C01810=1171.717,232.946,-63.644,-177.541,7.223,148.639
C01811=1171.722,232.698,-63.619,-177.544,7.221,148.640
C01812=1171.727,232.450,-63.593,-177.547,7.218,148.640
C01813=1171.731,232.200,-63.567,-177.549,7.216,148.640
C01814=1171.736,231.952,-63.541,-177.552,7.214,148.640
C01815=1171.740,231.703,-63.515,-177.555,7.211,148.640
C01816=1171.744,231.455,-63.489,-177.557,7.209,148.640
C01817=1171.749,231.207,-63.464,-177.560,7.206,148.640
C01818=1171.754,230.957,-63.437,-177.563,7.204,148.641
C01819=1171.758,230.709,-63.411,-177.566,7.201,148.641
C01820=1171.762,230.460,-63.386,-177.568,7.199,148.641
C01821=1171.767,230.212,-63.360,-177.571,7.196,148.641
C01822=1171.771,229.963,-63.335,-177.573,7.194,148.641
C01823=1171.775,229.714,-63.309,-177.576,7.192,148.642
C01824=1171.780,229.465,-63.282,-177.579,7.190,148.642
C01825=1171.785,229.217,-63.257,-177.581,7.187,148.642
C01826=1171.789,228.968,-63.231,-177.584,7.185,148.642
C01827=1171.794,228.719,-63.206,-177.587,7.182,148.642
C01828=1171.798,228.471,-63.180,-177.590,7.179,148.643
C01829=1171.803,228.222,-63.154,-177.592,7.177,148.643
C01830=1171.807,227.974,-63.129,-177.595,7.175,148.643
C01831=1171.812,227.725,-63.103,-177.598,7.172,148.643
C01832=1171.816,227.477,-63.078,-177.601,7.170,148.643
C01833=1171.820,227.228,-63.052,-177.603,7.168,148.644
C01834=1171.825,226.980,-63.026,-177.606,7.165,148.644
C01835=1171.829,226.731,-63.001,-177.609,7.163,148.644
C01836=1171.834,226.482,-62.974,-177.611,7.160,148.644
C01837=1171.839,226.234,-62.949,-177.614,7.158,148.644
C01838=1171.844,225.984,-62.924,-177.617,7.155,148.644
C01839=1171.848,225.735,-62.898,-177.619,7.153,148.645
C01840=1171.853,225.487,-62.873,-177.622,7.150,148.645
C01841=1171.857,225.239,-62.847,-177.625,7.149,148.645
C01842=1171.861,224.990,-62.821,-177.628,7.146,148.645
C01843=1171.866,224.742,-62.796,-177.630,7.144,148.646
C01844=1171.870,224.492,-62.771,-177.633,7.141,148.646
C01845=1171.875,224.243,-62.745,-177.636,7.139,148.646
C01846=1171.879,223.996,-62.720,-177.638,7.136,148.646
C01847=1171.883,223.747,-62.695,-177.641,7.134,148.646
C01848=1171.888,223.498,-62.670,-177.644,7.131,148.646
C01849=1171.892,223.249,-62.644,-177.646,7.130,148.647
C01850=1171.897,223.000,-62.618,-177.649,7.128,148.647
C01851=1171.901,222.752,-62.593,-177.651,7.125,148.647
C01852=1171.906,222.503,-62.568,-177.654,7.123,148.647
C01853=1171.911,222.255,-62.543,-177.657,7.120,148.647
C01854=1171.915,222.006,-62.517,-177.659,7.118,148.648
C01855=1171.920,221.757,-62.492,-177.662,7.115,148.648
C01856=1171.924,221.509,-62.466,-177.665,7.113,148.648
C01857=1171.928,221.260,-62.441,-177.668,7.110,148.648
C01858=1171.933,221.011,-62.417,-177.670,7.109,148.649
C01859=1171.937,220.763,-62.391,-177.674,7.106,148.649
C01860=1171.942,220.514,-62.366,-177.676,7.104,148.649
C01861=1171.946,220.265,-62.340,-177.679,7.101,148.649
C01862=1171.951,220.017,-62.315,-177.681,7.099,148.649
C01863=1171.955,219.768,-62.291,-177.684,7.096,148.650
C01864=1171.960,219.520,-62.265,-177.687,7.094,148.650
C01865=1171.964,219.270,-62.240,-177.689,7.093,148.650
C01866=1171.969,219.022,-62.215,-177.692,7.090,148.650
C01867=1171.974,218.773,-62.190,-177.695,7.088,148.651
C01868=1171.978,218.525,-62.165,-177.697,7.085,148.651
C01869=1171.982,218.275,-62.140,-177.700,7.083,148.651
C01870=1171.987,218.027,-62.115,-177.703,7.080,148.651
C01871=1171.992,217.778,-62.090,-177.706,7.078,148.651
C01872=1171.996,217.530,-62.065,-177.708,7.075,148.652
C01873=1172.000,217.281,-62.040,-177.711,7.074,148.652
C01874=1172.006,217.032,-62.015,-177.713,7.071,148.652
C01875=1172.010,216.783,-61.989,-177.716,7.069,148.652
C01876=1172.014,216.535,-61.965,-177.719,7.067,148.653
C01877=1172.018,216.286,-61.939,-177.722,7.064,148.653
C01878=1172.024,216.037,-61.915,-177.724,7.062,148.653
C01879=1172.027,215.788,-61.890,-177.727,7.059,148.653
C01880=1172.032,215.540,-61.865,-177.730,7.058,148.654
C01881=1172.037,215.291,-61.840,-177.732,7.055,148.654
C01882=1172.041,215.042,-61.816,-177.735,7.053,148.654
C01883=1172.045,214.793,-61.790,-177.738,7.051,148.654
C01884=1172.050,214.545,-61.765,-177.741,7.048,148.654
C01885=1172.055,214.296,-61.741,-177.743,7.046,148.655
C01886=1172.059,214.047,-61.716,-177.746,7.044,148.655
C01887=1172.064,213.799,-61.691,-177.749,7.042,148.655
C01888=1172.068,213.550,-61.666,-177.751,7.039,148.655
C01889=1172.073,213.301,-61.642,-177.754,7.037,148.656
C01890=1172.077,213.053,-61.617,-177.756,7.035,148.656
C01891=1172.082,212.804,-61.592,-177.759,7.033,148.656
C01892=1172.087,212.555,-61.567,-177.762,7.030,148.656
C01893=1172.091,212.306,-61.543,-177.765,7.028,148.656
C01894=1172.096,212.057,-61.518,-177.768,7.026,148.657
C01895=1172.100,211.809,-61.493,-177.770,7.023,148.657
C01896=1172.104,211.560,-61.468,-177.773,7.022,148.657
C01897=1172.109,211.312,-61.444,-177.776,7.019,148.658
C01898=1172.114,211.063,-61.420,-177.778,7.017,148.658
C01899=1172.118,210.813,-61.395,-177.781,7.014,148.658
C01900=1172.123,210.544,-61.368,-177.784,7.012,148.658
C01901=1172.128,210.273,-61.342,-177.787,7.010,148.658
C01902=1172.133,210.002,-61.315,-177.790,7.007,148.659
C01903=1172.138,209.732,-61.288,-177.793,7.005,148.659
C01904=1172.143,209.484,-61.263,-177.795,7.002,148.659
C01905=1172.147,209.234,-61.239,-177.798,7.000,148.659
C01906=1172.152,208.986,-61.214,-177.801,6.999,148.660
C01907=1172.156,208.737,-61.190,-177.804,6.996,148.660
C01908=1172.161,208.488,-61.165,-177.806,6.994,148.660
C01909=1172.165,208.239,-61.141,-177.809,6.991,148.660
C01910=1172.170,207.991,-61.116,-177.812,6.989,148.661
C01911=1172.175,207.742,-61.092,-177.814,6.987,148.661
C01912=1172.178,207.493,-61.068,-177.817,6.984,148.661
C01913=1172.184,207.245,-61.043,-177.820,6.983,148.661
C01914=1172.188,206.996,-61.019,-177.822,6.981,148.662
C01915=1172.192,206.747,-60.994,-177.825,6.978,148.662
C01916=1172.197,206.498,-60.970,-177.828,6.976,148.662
C01917=1172.202,206.249,-60.947,-177.830,6.974,148.662
C01918=1172.207,206.000,-60.922,-177.833,6.971,148.663
C01919=1172.210,205.751,-60.898,-177.836,6.970,148.663
C01920=1172.216,205.503,-60.873,-177.839,6.967,148.663
C01921=1172.220,205.254,-60.849,-177.841,6.965,148.663
C01922=1172.224,205.006,-60.825,-177.844,6.963,148.664
C01923=1172.230,204.757,-60.800,-177.847,6.960,148.664
C01924=1172.234,204.507,-60.776,-177.849,6.958,148.664
C01925=1172.238,204.259,-60.752,-177.852,6.956,148.664
C01926=1172.243,204.010,-60.728,-177.855,6.954,148.665
C01927=1172.248,203.762,-60.703,-177.858,6.952,148.665
C01928=1172.251,203.513,-60.679,-177.860,6.950,148.665
C01929=1172.256,203.264,-60.656,-177.863,6.947,148.665
C01930=1172.261,203.015,-60.631,-177.866,6.945,148.666
C01931=1172.266,202.767,-60.607,-177.868,6.943,148.666
C01932=1172.270,202.518,-60.583,-177.871,6.941,148.666
C01933=1172.275,202.268,-60.559,-177.874,6.939,148.667
C01934=1172.279,202.020,-60.534,-177.876,6.937,148.667
C01935=1172.284,201.771,-60.510,-177.879,6.934,148.667
C01936=1172.288,201.522,-60.487,-177.882,6.932,148.667
C01937=1172.293,201.274,-60.463,-177.884,6.930,148.668
C01938=1172.298,201.025,-60.438,-177.887,6.928,148.668
C01939=1172.302,200.775,-60.415,-177.890,6.926,148.668
C01940=1172.306,200.527,-60.391,-177.892,6.924,148.668
C01941=1172.311,200.279,-60.366,-177.895,6.921,148.669
C01942=1172.315,200.030,-60.343,-177.898,6.919,148.669
C01943=1172.321,199.781,-60.318,-177.901,6.918,148.669
C01944=1172.325,199.532,-60.295,-177.903,6.915,148.669
C01945=1172.330,199.283,-60.271,-177.906,6.913,148.670
C01946=1172.334,199.034,-60.248,-177.909,6.911,148.670
C01947=1172.338,198.785,-60.223,-177.911,6.909,148.670
C01948=1172.343,198.537,-60.199,-177.914,6.906,148.671
C01949=1172.347,198.288,-60.176,-177.917,6.905,148.671
C01950=1172.352,198.039,-60.151,-177.919,6.902,148.671
C01951=1172.357,197.790,-60.128,-177.922,6.900,148.671
C01952=1172.361,197.542,-60.104,-177.925,6.898,148.672
C01953=1172.366,197.293,-60.080,-177.927,6.896,148.672
C01954=1172.371,197.044,-60.057,-177.930,6.894,148.672
C01955=1172.375,196.795,-60.033,-177.933,6.892,148.673
C01956=1172.380,196.546,-60.009,-177.936,6.890,148.673
C01957=1172.384,196.298,-59.985,-177.938,6.888,148.673
C01958=1172.389,196.049,-59.962,-177.941,6.885,148.673
C01959=1172.393,195.800,-59.938,-177.944,6.883,148.674
C01960=1172.398,195.550,-59.914,-177.946,6.881,148.674
C01961=1172.402,195.301,-59.891,-177.949,6.879,148.674
C01962=1172.407,195.053,-59.867,-177.952,6.877,148.675
C01963=1172.411,194.804,-59.843,-177.955,6.875,148.675
C01964=1172.416,194.555,-59.820,-177.957,6.873,148.675
C01965=1172.420,194.307,-59.796,-177.960,6.870,148.675
C01966=1172.425,194.058,-59.773,-177.963,6.869,148.676
C01967=1172.430,193.808,-59.749,-177.966,6.867,148.676
C01968=1172.434,193.560,-59.725,-177.968,6.865,148.676
C01969=1172.439,193.311,-59.702,-177.971,6.862,148.676
C01970=1172.444,193.062,-59.679,-177.974,6.860,148.677
C01971=1172.448,192.814,-59.654,-177.976,6.858,148.677
C01972=1172.453,192.565,-59.631,-177.979,6.856,148.677
C01973=1172.457,192.316,-59.608,-177.982,6.854,148.678
C01974=1172.462,192.066,-59.584,-177.985,6.852,148.678
C01975=1172.466,191.818,-59.560,-177.987,6.850,148.678
C01976=1172.471,191.569,-59.537,-177.989,6.848,148.679
C01977=1172.476,191.320,-59.514,-177.993,6.845,148.679
C01978=1172.481,191.071,-59.490,-177.995,6.844,148.679
C01979=1172.486,190.823,-59.467,-177.997,6.842,148.679
C01980=1172.491,190.574,-59.444,-178.000,6.840,148.680
C01981=1172.495,190.325,-59.420,-178.003,6.837,148.680
C01982=1172.499,190.077,-59.397,-178.006,6.835,148.680
C01983=1172.504,189.827,-59.374,-178.009,6.834,148.681
C01984=1172.508,189.578,-59.350,-178.011,6.832,148.681
C01985=1172.513,189.329,-59.327,-178.014,6.829,148.681
C01986=1172.518,189.080,-59.304,-178.017,6.827,148.682
C01987=1172.522,188.831,-59.280,-178.020,6.825,148.682
C01988=1172.527,188.582,-59.257,-178.022,6.823,148.682
C01989=1172.531,188.334,-59.234,-178.024,6.822,148.682
C01990=1172.536,188.085,-59.211,-178.028,6.819,148.683
C01991=1172.541,187.836,-59.188,-178.030,6.817,148.683
C01992=1172.546,187.587,-59.164,-178.033,6.815,148.683
C01993=1172.551,187.338,-59.141,-178.035,6.813,148.684
C01994=1172.554,187.089,-59.118,-178.038,6.811,148.684
C01995=1172.559,186.840,-59.095,-178.041,6.809,148.684
C01996=1172.564,186.591,-59.072,-178.044,6.807,148.685
C01997=1172.569,186.342,-59.048,-178.046,6.805,148.685
C01998=1172.573,186.094,-59.025,-178.049,6.803,148.685
C01999=1172.578,185.845,-59.002,-178.052,6.801,148.685
C02000=1172.583,185.596,-58.979,-178.055,6.799,148.686
C02001=1172.587,185.347,-58.956,-178.057,6.797,148.686
C02002=1172.591,185.098,-58.933,-178.060,6.795,148.686
C02003=1172.596,184.849,-58.910,-178.063,6.792,148.687
C02004=1172.601,184.580,-58.885,-178.065,6.791,148.687
C02005=1172.606,184.310,-58.860,-178.068,6.789,148.687
C02006=1172.611,184.040,-58.835,-178.071,6.786,148.688
C02007=1172.616,183.771,-58.810,-178.074,6.784,148.688
C02008=1172.620,183.522,-58.787,-178.077,6.782,148.688
C02009=1172.625,183.273,-58.764,-178.080,6.780,148.689
C02010=1172.630,183.025,-58.741,-178.082,6.778,148.689
C02011=1172.634,182.776,-58.718,-178.085,6.776,148.689
C02012=1172.639,182.526,-58.696,-178.088,6.774,148.690
C02013=1172.643,182.278,-58.673,-178.090,6.773,148.690
C02014=1172.648,182.029,-58.649,-178.093,6.770,148.690
C02015=1172.653,181.780,-58.626,-178.096,6.768,148.691
C02016=1172.658,181.531,-58.604,-178.098,6.766,148.691
C02017=1172.662,181.282,-58.581,-178.101,6.764,148.691
C02018=1172.666,181.033,-58.558,-178.104,6.763,148.691
C02019=1172.672,180.785,-58.535,-178.107,6.760,148.692
C02020=1172.677,180.535,-58.513,-178.110,6.758,148.692
C02021=1172.681,180.286,-58.490,-178.112,6.757,148.693
C02022=1172.685,180.037,-58.466,-178.115,6.754,148.693
C02023=1172.690,179.789,-58.445,-178.117,6.753,148.693
C02024=1172.695,179.540,-58.421,-178.120,6.751,148.693
C02025=1172.699,179.291,-58.399,-178.123,6.748,148.694
C02026=1172.704,179.041,-58.376,-178.126,6.747,148.694
C02027=1172.708,178.793,-58.354,-178.129,6.745,148.694
C02028=1172.713,178.544,-58.331,-178.131,6.743,148.695
C02029=1172.717,178.295,-58.308,-178.133,6.741,148.695
C02030=1172.723,178.047,-58.285,-178.136,6.739,148.695
C02031=1172.727,177.797,-58.263,-178.139,6.737,148.696
C02032=1172.732,177.548,-58.240,-178.142,6.735,148.696
C02033=1172.736,177.300,-58.218,-178.145,6.733,148.696
C02034=1172.741,177.051,-58.195,-178.147,6.731,148.697
C02035=1172.745,176.801,-58.173,-178.150,6.729,148.697
C02036=1172.750,176.552,-58.149,-178.152,6.727,148.697
C02037=1172.755,176.304,-58.128,-178.155,6.726,148.698
C02038=1172.760,176.054,-58.104,-178.158,6.723,148.698
C02039=1172.765,175.806,-58.083,-178.161,6.721,148.698
C02040=1172.768,175.557,-58.060,-178.164,6.719,148.699
C02041=1172.774,175.307,-58.037,-178.166,6.718,148.699
C02042=1172.778,175.059,-58.015,-178.169,6.716,148.699
C02043=1172.783,174.810,-57.992,-178.171,6.714,148.700
C02044=1172.787,174.560,-57.970,-178.174,6.712,148.700
C02045=1172.792,174.312,-57.948,-178.177,6.710,148.700
C02046=1172.797,174.063,-57.925,-178.180,6.708,148.701
C02047=1172.801,173.814,-57.902,-178.182,6.706,148.701
C02048=1172.806,173.565,-57.881,-178.185,6.704,148.701
C02049=1172.811,173.316,-57.858,-178.188,6.702,148.702
C02050=1172.815,173.068,-57.836,-178.190,6.701,148.702
C02051=1172.820,172.818,-57.813,-178.193,6.699,148.702
C02052=1172.825,172.569,-57.791,-178.195,6.697,148.703
C02053=1172.829,172.321,-57.769,-178.198,6.695,148.703
C02054=1172.834,172.071,-57.746,-178.201,6.692,148.703
C02055=1172.839,171.822,-57.724,-178.204,6.691,148.704
C02056=1172.843,171.574,-57.701,-178.207,6.689,148.704
C02057=1172.847,171.324,-57.679,-178.209,6.687,148.704
C02058=1172.853,171.075,-57.657,-178.212,6.685,148.705
C02059=1172.857,170.826,-57.635,-178.215,6.684,148.705
C02060=1172.862,170.578,-57.613,-178.217,6.682,148.705
C02061=1172.867,170.328,-57.590,-178.220,6.680,148.706
C02062=1172.872,170.080,-57.568,-178.222,6.678,148.706
C02063=1172.876,169.830,-57.546,-178.226,6.675,148.706
C02064=1172.881,169.582,-57.525,-178.228,6.674,148.707
C02065=1172.885,169.333,-57.502,-178.231,6.672,148.707
C02066=1172.890,169.084,-57.480,-178.234,6.670,148.707
C02067=1172.895,168.835,-57.458,-178.236,6.668,148.708
C02068=1172.899,168.586,-57.436,-178.239,6.667,148.708
C02069=1172.904,168.337,-57.414,-178.242,6.665,148.709
C02070=1172.909,168.088,-57.392,-178.244,6.663,148.709
C02071=1172.914,167.839,-57.369,-178.247,6.661,148.709
C02072=1172.918,167.590,-57.348,-178.250,6.659,148.710
C02073=1172.922,167.341,-57.325,-178.252,6.658,148.710
C02074=1172.927,167.093,-57.303,-178.255,6.656,148.710
C02075=1172.932,166.843,-57.281,-178.258,6.653,148.711
C02076=1172.937,166.594,-57.259,-178.261,6.651,148.711
C02077=1172.941,166.345,-57.237,-178.263,6.650,148.711
C02078=1172.946,166.096,-57.215,-178.266,6.648,148.712
C02079=1172.951,165.847,-57.193,-178.269,6.646,148.712
C02080=1172.955,165.598,-57.172,-178.271,6.644,148.712
C02081=1172.960,165.349,-57.150,-178.274,6.642,148.713
C02082=1172.965,165.100,-57.128,-178.277,6.641,148.713
C02083=1172.969,164.851,-57.106,-178.279,6.639,148.713
C02084=1172.974,164.602,-57.084,-178.282,6.637,148.714
C02085=1172.979,164.353,-57.061,-178.285,6.635,148.714
C02086=1172.984,164.104,-57.040,-178.287,6.634,148.715
C02087=1172.988,163.855,-57.018,-178.290,6.632,148.715
C02088=1172.993,163.606,-56.996,-178.293,6.630,148.715
C02089=1172.998,163.357,-56.975,-178.296,6.628,148.716
C02090=1173.002,163.107,-56.953,-178.298,6.627,148.716
C02091=1173.007,162.859,-56.931,-178.301,6.625,148.716
C02092=1173.012,162.610,-56.910,-178.304,6.622,148.717
C02093=1173.016,162.361,-56.888,-178.307,6.621,148.717
C02094=1173.021,162.112,-56.866,-178.310,6.619,148.718
C02095=1173.025,161.863,-56.844,-178.312,6.617,148.718
C02096=1173.030,161.614,-56.822,-178.315,6.615,148.718
C02097=1173.035,161.365,-56.801,-178.318,6.613,148.719
C02098=1173.040,161.116,-56.779,-178.320,6.612,148.719
C02099=1173.044,160.867,-56.758,-178.323,6.610,148.719
C02100=1173.049,160.618,-56.735,-178.325,6.608,148.720
C02101=1173.054,160.369,-56.714,-178.328,6.606,148.720
C02102=1173.059,160.120,-56.693,-178.331,6.604,148.720
C02103=1173.063,159.870,-56.671,-178.333,6.603,148.721
C02104=1173.067,159.622,-56.650,-178.336,6.601,148.721
C02105=1173.072,159.373,-56.628,-178.339,6.599,148.721
C02106=1173.077,159.123,-56.607,-178.341,6.597,148.722
C02107=1173.081,158.875,-56.585,-178.344,6.596,148.722
C02108=1173.087,158.605,-56.562,-178.347,6.594,148.723
C02109=1173.091,158.337,-56.538,-178.350,6.592,148.723
C02110=1173.097,158.068,-56.515,-178.353,6.590,148.723
C02111=1173.102,157.799,-56.492,-178.356,6.588,148.724
C02112=1173.106,157.550,-56.470,-178.358,6.586,148.724
C02113=1173.112,157.301,-56.449,-178.361,6.585,148.725
C02114=1173.116,157.051,-56.427,-178.364,6.583,148.725
C02115=1173.121,156.803,-56.406,-178.367,6.581,148.725
C02116=1173.126,156.553,-56.385,-178.369,6.579,148.726
C02117=1173.130,156.305,-56.364,-178.372,6.578,148.726
C02118=1173.135,156.055,-56.342,-178.375,6.576,148.727
C02119=1173.140,155.807,-56.321,-178.377,6.574,148.727
C02120=1173.145,155.557,-56.300,-178.380,6.572,148.727
C02121=1173.149,155.308,-56.278,-178.383,6.571,148.728
C02122=1173.153,155.060,-56.256,-178.385,6.569,148.728
C02123=1173.158,154.810,-56.236,-178.388,6.567,148.728
C02124=1173.163,154.562,-56.214,-178.391,6.565,148.729
C02125=1173.168,154.312,-56.192,-178.393,6.564,148.729
C02126=1173.173,154.063,-56.171,-178.396,6.562,148.730
C02127=1173.177,153.814,-56.150,-178.399,6.560,148.730
C02128=1173.182,153.565,-56.129,-178.402,6.558,148.730
C02129=1173.187,153.316,-56.108,-178.404,6.556,148.731
C02130=1173.192,153.066,-56.086,-178.407,6.555,148.731
C02131=1173.196,152.818,-56.065,-178.410,6.553,148.731
C02132=1173.201,152.569,-56.044,-178.412,6.551,148.732
C02133=1173.206,152.320,-56.023,-178.415,6.550,148.732
C02134=1173.210,152.071,-56.002,-178.418,6.548,148.733
C02135=1173.215,151.822,-55.980,-178.421,6.546,148.733
C02136=1173.220,151.572,-55.959,-178.424,6.545,148.734
C02137=1173.225,151.323,-55.938,-178.426,6.543,148.734
C02138=1173.229,151.075,-55.917,-178.429,6.541,148.734
C02139=1173.234,150.826,-55.896,-178.432,6.539,148.735
C02140=1173.239,150.576,-55.875,-178.434,6.538,148.735
C02141=1173.243,150.327,-55.854,-178.437,6.536,148.735
C02142=1173.248,150.078,-55.833,-178.440,6.534,148.736
C02143=1173.253,149.829,-55.812,-178.442,6.533,148.736
C02144=1173.257,149.581,-55.791,-178.445,6.531,148.737
C02145=1173.263,149.331,-55.770,-178.447,6.530,148.737
C02146=1173.267,149.082,-55.750,-178.450,6.528,148.737
C02147=1173.272,148.832,-55.728,-178.453,6.526,148.738
C02148=1173.276,148.584,-55.707,-178.455,6.524,148.738
C02149=1173.281,148.335,-55.686,-178.458,6.523,148.738
C02150=1173.286,148.085,-55.665,-178.461,6.521,148.739
C02151=1173.291,147.837,-55.645,-178.463,6.519,148.739
C02152=1173.295,147.588,-55.623,-178.467,6.518,148.740
C02153=1173.301,147.339,-55.602,-178.469,6.516,148.740
C02154=1173.305,147.090,-55.582,-178.472,6.514,148.741
C02155=1173.310,146.840,-55.560,-178.475,6.512,148.741
C02156=1173.314,146.591,-55.540,-178.477,6.511,148.741
C02157=1173.319,146.342,-55.519,-178.480,6.509,148.742
C02158=1173.323,146.093,-55.498,-178.483,6.507,148.742
C02159=1173.328,145.844,-55.477,-178.485,6.505,148.743
C02160=1173.333,145.595,-55.457,-178.488,6.505,148.743
C02161=1173.338,145.346,-55.436,-178.490,6.503,148.743
C02162=1173.343,145.097,-55.415,-178.493,6.501,148.744
C02163=1173.348,144.848,-55.394,-178.496,6.499,148.744
C02164=1173.352,144.599,-55.374,-178.499,6.498,148.745
C02165=1173.357,144.349,-55.353,-178.502,6.496,148.745
C02166=1173.362,144.100,-55.333,-178.504,6.494,148.745
C02167=1173.367,143.851,-55.312,-178.507,6.493,148.746
C02168=1173.371,143.601,-55.291,-178.510,6.491,148.746
C02169=1173.376,143.353,-55.269,-178.512,6.489,148.747
C02170=1173.380,143.104,-55.249,-178.515,6.487,148.747
C02171=1173.385,142.855,-55.229,-178.518,6.486,148.747
C02172=1173.390,142.606,-55.208,-178.520,6.485,148.748
C02173=1173.394,142.357,-55.187,-178.523,6.483,148.748
C02174=1173.400,142.107,-55.167,-178.526,6.482,148.749
C02175=1173.404,141.858,-55.147,-178.528,6.480,148.749
C02176=1173.409,141.609,-55.126,-178.531,6.478,148.750
C02177=1173.414,141.360,-55.105,-178.534,6.476,148.750
C02178=1173.418,141.111,-55.085,-178.536,6.475,148.750
C02179=1173.423,140.861,-55.064,-178.539,6.473,148.751
C02180=1173.428,140.612,-55.044,-178.542,6.471,148.751
C02181=1173.432,140.364,-55.023,-178.544,6.470,148.751
C02182=1173.437,140.114,-55.002,-178.547,6.468,148.752
C02183=1173.442,139.865,-54.982,-178.550,6.467,148.752
C02184=1173.446,139.616,-54.961,-178.553,6.465,148.753
C02185=1173.452,139.367,-54.941,-178.555,6.464,148.753
C02186=1173.456,139.118,-54.921,-178.558,6.462,148.754
C02187=1173.461,138.869,-54.900,-178.561,6.460,148.754
C02188=1173.466,138.620,-54.880,-178.563,6.458,148.754
C02189=1173.471,138.371,-54.859,-178.566,6.457,148.755
C02190=1173.475,138.122,-54.839,-178.568,6.456,148.755
C02191=1173.481,137.872,-54.819,-178.571,6.454,148.756
C02192=1173.485,137.623,-54.798,-178.574,6.453,148.756
C02193=1173.490,137.374,-54.778,-178.577,6.451,148.757
C02194=1173.494,137.125,-54.758,-178.579,6.449,148.757
C02195=1173.499,136.876,-54.737,-178.582,6.447,148.757
C02196=1173.504,136.627,-54.717,-178.585,6.446,148.758
C02197=1173.508,136.378,-54.697,-178.587,6.445,148.758
C02198=1173.513,136.129,-54.676,-178.590,6.443,148.759
C02199=1173.518,135.879,-54.656,-178.593,6.442,148.759
C02200=1173.523,135.631,-54.636,-178.596,6.440,148.760
C02201=1173.528,135.382,-54.616,-178.598,6.438,148.760
C02202=1173.532,135.132,-54.596,-178.601,6.436,148.760
C02203=1173.537,134.883,-54.576,-178.604,6.435,148.761
C02204=1173.542,134.634,-54.555,-178.606,6.434,148.761
C02205=1173.547,134.384,-54.535,-178.609,6.432,148.762
C02206=1173.551,134.135,-54.515,-178.612,6.431,148.762
C02207=1173.556,133.886,-54.494,-178.614,6.429,148.763
C02208=1173.561,133.638,-54.475,-178.617,6.427,148.763
C02209=1173.566,133.388,-54.454,-178.620,6.425,148.763
C02210=1173.571,133.139,-54.434,-178.622,6.424,148.764
C02211=1173.575,132.890,-54.414,-178.625,6.423,148.764
C02212=1173.580,132.621,-54.393,-178.628,6.421,148.765
C02213=1173.586,132.353,-54.371,-178.630,6.419,148.765
C02214=1173.591,132.084,-54.349,-178.634,6.418,148.766
C02215=1173.596,131.815,-54.328,-178.637,6.416,148.766
C02216=1173.601,131.566,-54.307,-178.639,6.415,148.766
C02217=1173.605,131.317,-54.288,-178.642,6.413,148.767
C02218=1173.610,131.068,-54.268,-178.645,6.412,148.767
C02219=1173.615,130.819,-54.248,-178.648,6.410,148.768
C02220=1173.620,130.570,-54.228,-178.650,6.408,148.768
C02221=1173.624,130.320,-54.208,-178.652,6.407,148.769
C02222=1173.629,130.071,-54.188,-178.655,6.405,148.769
C02223=1173.634,129.822,-54.168,-178.658,6.404,148.769
C02224=1173.639,129.574,-54.148,-178.661,6.402,148.770
C02225=1173.644,129.324,-54.128,-178.664,6.401,148.770
C02226=1173.649,129.074,-54.108,-178.666,6.399,148.771
C02227=1173.654,128.826,-54.088,-178.669,6.398,148.771
C02228=1173.659,128.576,-54.068,-178.671,6.396,148.772
C02229=1173.663,128.327,-54.048,-178.675,6.395,148.772
C02230=1173.668,128.078,-54.028,-178.677,6.393,148.773
C02231=1173.673,127.829,-54.009,-178.680,6.391,148.773
C02232=1173.678,127.580,-53.989,-178.682,6.390,148.773
C02233=1173.682,127.330,-53.969,-178.685,6.389,148.774
C02234=1173.687,127.081,-53.949,-178.688,6.387,148.774
C02235=1173.691,126.833,-53.930,-178.691,6.385,148.775
C02236=1173.696,126.583,-53.910,-178.693,6.384,148.775
C02237=1173.701,126.334,-53.891,-178.695,6.383,148.776
C02238=1173.705,126.085,-53.870,-178.698,6.381,148.776
C02239=1173.711,125.836,-53.851,-178.701,6.380,148.777
C02240=1173.715,125.586,-53.831,-178.704,6.378,148.777
C02241=1173.720,125.337,-53.812,-178.707,6.376,148.777
C02242=1173.725,125.089,-53.792,-178.709,6.375,148.778
C02243=1173.730,124.839,-53.772,-178.712,6.374,148.778
C02244=1173.735,124.589,-53.752,-178.715,6.372,148.779
C02245=1173.739,124.340,-53.733,-178.717,6.370,148.779
C02246=1173.745,124.091,-53.714,-178.720,6.370,148.780
C02247=1173.748,123.842,-53.694,-178.722,6.368,148.780
C02248=1173.753,123.593,-53.674,-178.726,6.366,148.781
C02249=1173.758,123.344,-53.655,-178.728,6.365,148.781
C02250=1173.763,123.094,-53.635,-178.730,6.364,148.782
C02251=1173.768,122.845,-53.615,-178.733,6.362,148.782
C02252=1173.773,122.596,-53.596,-178.736,6.360,148.782
C02253=1173.778,122.347,-53.576,-178.739,6.359,148.783
C02254=1173.782,122.098,-53.557,-178.742,6.357,148.783
C02255=1173.787,121.849,-53.537,-178.744,6.356,148.784
C02256=1173.792,121.599,-53.518,-178.746,6.355,148.784
C02257=1173.797,121.350,-53.499,-178.750,6.353,148.785
C02258=1173.802,121.101,-53.479,-178.752,6.351,148.785
C02259=1173.806,120.852,-53.460,-178.755,6.351,148.786
C02260=1173.811,120.603,-53.441,-178.757,6.349,148.786
C02261=1173.816,120.353,-53.421,-178.760,6.347,148.787
C02262=1173.821,120.104,-53.402,-178.763,6.346,148.787
C02263=1173.826,119.855,-53.382,-178.765,6.345,148.787
C02264=1173.830,119.605,-53.363,-178.768,6.343,148.788
C02265=1173.835,119.357,-53.344,-178.771,6.342,148.788
C02266=1173.840,119.107,-53.324,-178.774,6.340,148.789
C02267=1173.846,118.858,-53.305,-178.776,6.339,148.789
C02268=1173.850,118.609,-53.286,-178.779,6.337,148.790
C02269=1173.854,118.359,-53.266,-178.782,6.336,148.790
C02270=1173.860,118.110,-53.247,-178.785,6.334,148.791
C02271=1173.864,117.861,-53.228,-178.787,6.333,148.791
C02272=1173.869,117.612,-53.208,-178.789,6.332,148.792
C02273=1173.874,117.363,-53.189,-178.793,6.330,148.792
C02274=1173.879,117.114,-53.169,-178.795,6.329,148.793
C02275=1173.883,116.865,-53.150,-178.797,6.328,148.793
C02276=1173.888,116.616,-53.131,-178.800,6.326,148.793
C02277=1173.893,116.366,-53.111,-178.803,6.324,148.794
C02278=1173.897,116.116,-53.093,-178.805,6.324,148.794
C02279=1173.903,115.867,-53.074,-178.808,6.322,148.795
C02280=1173.908,115.618,-53.054,-178.811,6.320,148.795
C02281=1173.912,115.369,-53.035,-178.814,6.320,148.796
C02282=1173.917,115.120,-53.016,-178.816,6.318,148.796
C02283=1173.922,114.871,-52.996,-178.819,6.316,148.797
C02284=1173.927,114.621,-52.978,-178.822,6.315,148.797
C02285=1173.932,114.372,-52.959,-178.824,6.314,148.798
C02286=1173.936,114.123,-52.940,-178.827,6.312,148.798
C02287=1173.941,113.874,-52.920,-178.830,6.310,148.798
C02288=1173.946,113.624,-52.901,-178.832,6.310,148.799
C02289=1173.951,113.375,-52.883,-178.835,6.308,148.800
C02290=1173.956,113.126,-52.863,-178.838,6.306,148.800
C02291=1173.960,112.877,-52.844,-178.840,6.305,148.800
C02292=1173.966,112.628,-52.826,-178.843,6.304,148.801
C02293=1173.970,112.378,-52.807,-178.846,6.302,148.801
C02294=1173.975,112.130,-52.787,-178.848,6.301,148.802
C02295=1173.980,111.880,-52.768,-178.851,6.300,148.802
C02296=1173.985,111.631,-52.750,-178.854,6.298,148.803
C02297=1173.990,111.381,-52.730,-178.856,6.297,148.803
C02298=1173.994,111.133,-52.711,-178.859,6.296,148.804
C02299=1173.999,110.882,-52.693,-178.862,6.294,148.804
C02300=1174.004,110.634,-52.674,-178.865,6.293,148.805
C02301=1174.009,110.385,-52.655,-178.867,6.292,148.805
C02302=1174.014,110.135,-52.636,-178.870,6.290,148.806
C02303=1174.019,109.886,-52.617,-178.873,6.289,148.806
C02304=1174.023,109.636,-52.599,-178.875,6.288,148.807
C02305=1174.029,109.388,-52.579,-178.878,6.286,148.807
C02306=1174.033,109.138,-52.560,-178.881,6.285,148.808
C02307=1174.037,108.889,-52.542,-178.883,6.283,148.808
C02308=1174.043,108.640,-52.523,-178.886,6.282,148.809
C02309=1174.047,108.390,-52.505,-178.889,6.281,148.809
C02310=1174.052,108.142,-52.485,-178.891,6.279,148.809
C02311=1174.057,107.892,-52.467,-178.893,6.278,148.810
C02312=1174.062,107.643,-52.448,-178.897,6.277,148.810
C02313=1174.067,107.394,-52.430,-178.899,6.275,148.811
C02314=1174.071,107.144,-52.411,-178.902,6.274,148.811
C02315=1174.077,106.895,-52.392,-178.905,6.273,148.812
C02316=1174.081,106.627,-52.372,-178.907,6.271,148.812
C02317=1174.087,106.358,-52.352,-178.911,6.269,148.813
C02318=1174.093,106.089,-52.332,-178.913,6.269,148.813
C02319=1174.097,105.822,-52.311,-178.916,6.267,148.814
C02320=1174.102,105.573,-52.293,-178.919,6.265,148.814
C02321=1174.107,105.323,-52.274,-178.921,6.264,148.815
C02322=1174.112,105.074,-52.256,-178.924,6.263,148.815
C02323=1174.118,104.824,-52.237,-178.927,6.261,148.816
C02324=1174.122,104.575,-52.218,-178.929,6.260,148.816
C02325=1174.126,104.326,-52.200,-178.932,6.259,148.817
C02326=1174.132,104.077,-52.181,-178.935,6.258,148.817
C02327=1174.136,103.827,-52.163,-178.937,6.257,148.818
C02328=1174.141,103.578,-52.145,-178.940,6.255,148.818
C02329=1174.146,103.329,-52.126,-178.943,6.254,148.819
C02330=1174.151,103.079,-52.107,-178.945,6.253,148.819
C02331=1174.156,102.830,-52.089,-178.948,6.251,148.820
C02332=1174.160,102.582,-52.070,-178.951,6.250,148.820
C02333=1174.166,102.332,-52.052,-178.953,6.249,148.821
C02334=1174.170,102.082,-52.033,-178.956,6.247,148.821
C02335=1174.175,101.834,-52.015,-178.958,6.246,148.822
C02336=1174.180,101.584,-51.997,-178.961,6.245,148.822
C02337=1174.185,101.334,-51.978,-178.964,6.243,148.823
C02338=1174.190,101.085,-51.960,-178.966,6.242,148.823
C02339=1174.194,100.836,-51.941,-178.969,6.241,148.824
C02340=1174.199,100.587,-51.923,-178.972,6.239,148.824
C02341=1174.204,100.337,-51.904,-178.974,6.238,148.825
C02342=1174.209,100.088,-51.886,-178.977,6.237,148.825
C02343=1174.214,99.839,-51.868,-178.980,6.236,148.826
C02344=1174.219,99.590,-51.849,-178.982,6.234,148.826
C02345=1174.224,99.341,-51.832,-178.986,6.233,148.827
C02346=1174.229,99.091,-51.813,-178.988,6.232,148.827
C02347=1174.233,98.842,-51.795,-178.991,6.230,148.828
C02348=1174.238,98.592,-51.777,-178.993,6.230,148.828
C02349=1174.243,98.343,-51.759,-178.996,6.228,148.829
C02350=1174.247,98.094,-51.740,-178.999,6.226,148.829
C02351=1174.252,97.845,-51.722,-179.001,6.226,148.830
C02352=1174.257,97.596,-51.704,-179.004,6.224,148.830
C02353=1174.263,97.346,-51.685,-179.006,6.223,148.831
C02354=1174.268,97.097,-51.667,-179.009,6.222,148.831
C02355=1174.272,96.847,-51.649,-179.012,6.220,148.832
C02356=1174.277,96.598,-51.631,-179.015,6.220,148.832
C02357=1174.282,96.349,-51.613,-179.017,6.218,148.833
C02358=1174.287,96.100,-51.595,-179.019,6.217,148.833
C02359=1174.292,95.850,-51.577,-179.023,6.216,148.834
C02360=1174.297,95.601,-51.559,-179.025,6.214,148.834
C02361=1174.301,95.351,-51.540,-179.028,6.213,148.835
C02362=1174.307,95.102,-51.522,-179.031,6.212,148.835
C02363=1174.311,94.853,-51.504,-179.033,6.211,148.836
C02364=1174.316,94.604,-51.486,-179.036,6.209,148.836
C02365=1174.321,94.354,-51.468,-179.038,6.209,148.837
C02366=1174.326,94.105,-51.450,-179.041,6.207,148.837
C02367=1174.331,93.856,-51.432,-179.044,6.206,148.838
C02368=1174.335,93.606,-51.414,-179.046,6.205,148.838
C02369=1174.340,93.357,-51.396,-179.049,6.203,148.839
C02370=1174.345,93.108,-51.378,-179.052,6.202,148.839
C02371=1174.350,92.859,-51.360,-179.054,6.201,148.840
C02372=1174.355,92.609,-51.342,-179.057,6.200,148.840
C02373=1174.360,92.360,-51.324,-179.060,6.198,148.841
C02374=1174.365,92.111,-51.306,-179.062,6.197,148.841
C02375=1174.370,91.862,-51.288,-179.065,6.196,148.842
C02376=1174.375,91.613,-51.270,-179.068,6.194,148.842
C02377=1174.380,91.363,-51.253,-179.070,6.194,148.843
C02378=1174.384,91.113,-51.234,-179.073,6.192,148.843
C02379=1174.389,90.864,-51.216,-179.075,6.191,148.844
C02380=1174.394,90.615,-51.198,-179.078,6.190,148.844
C02381=1174.399,90.366,-51.180,-179.081,6.189,148.845
C02382=1174.404,90.116,-51.162,-179.084,6.188,148.845
C02383=1174.409,89.867,-51.145,-179.086,6.186,148.846
C02384=1174.413,89.618,-51.128,-179.089,6.185,148.846
C02385=1174.418,89.369,-51.110,-179.092,6.184,148.847
C02386=1174.423,89.119,-51.092,-179.094,6.183,148.847
C02387=1174.428,88.870,-51.074,-179.097,6.181,148.848
C02388=1174.433,88.620,-51.056,-179.099,6.181,148.848
C02389=1174.438,88.371,-51.038,-179.102,6.179,148.849
C02390=1174.443,88.122,-51.020,-179.105,6.178,148.849
C02391=1174.448,87.873,-51.002,-179.107,6.177,148.850
C02392=1174.453,87.623,-50.985,-179.110,6.176,148.851
C02393=1174.457,87.374,-50.968,-179.113,6.174,148.851
C02394=1174.462,87.125,-50.950,-179.115,6.174,148.852
C02395=1174.467,86.875,-50.933,-179.118,6.172,148.852
C02396=1174.472,86.626,-50.915,-179.120,6.171,148.852
C02397=1174.477,86.377,-50.897,-179.123,6.170,148.853
C02398=1174.483,86.127,-50.879,-179.126,6.168,148.854
C02399=1174.487,85.878,-50.861,-179.129,6.168,148.854
C02400=1174.492,85.629,-50.844,-179.131,6.166,148.855
C02401=1174.497,85.379,-50.827,-179.134,6.165,148.855
C02402=1174.502,85.130,-50.809,-179.137,6.164,148.856
C02403=1174.507,84.881,-50.791,-179.139,6.163,148.856
C02404=1174.512,84.631,-50.774,-179.142,6.161,148.857
C02405=1174.516,84.382,-50.756,-179.144,6.161,148.857
C02406=1174.521,84.132,-50.739,-179.148,6.159,148.858
C02407=1174.526,83.883,-50.721,-179.150,6.158,148.858
C02408=1174.531,83.633,-50.704,-179.152,6.157,148.859
C02409=1174.536,83.385,-50.686,-179.155,6.156,148.859
C02410=1174.540,83.135,-50.668,-179.158,6.154,148.860
C02411=1174.546,82.886,-50.651,-179.160,6.154,148.860
C02412=1174.551,82.636,-50.633,-179.163,6.152,148.861
C02413=1174.555,82.387,-50.616,-179.166,6.152,148.861
C02414=1174.560,82.138,-50.598,-179.168,6.150,148.862
C02415=1174.565,81.888,-50.581,-179.171,6.149,148.862
C02416=1174.570,81.640,-50.564,-179.174,6.148,148.863
C02417=1174.575,81.390,-50.547,-179.176,6.147,148.863
C02418=1174.580,81.141,-50.529,-179.179,6.145,148.864
C02419=1174.585,80.891,-50.512,-179.181,6.145,148.864
C02420=1174.590,80.623,-50.493,-179.185,6.143,148.865
C02421=1174.595,80.354,-50.474,-179.187,6.143,148.866
C02422=1174.601,80.086,-50.456,-179.190,6.141,148.866
C02423=1174.606,79.817,-50.437,-179.193,6.140,148.867
C02424=1174.611,79.568,-50.420,-179.195,6.139,148.867
C02425=1174.616,79.319,-50.402,-179.198,6.137,148.868
C02426=1174.620,79.069,-50.386,-179.201,6.137,148.868
C02427=1174.626,78.821,-50.368,-179.204,6.135,148.869
C02428=1174.631,78.571,-50.351,-179.206,6.134,148.869
C02429=1174.635,78.322,-50.333,-179.209,6.133,148.870
C02430=1174.640,78.072,-50.316,-179.211,6.132,148.870
C02431=1174.646,77.822,-50.299,-179.214,6.130,148.871
C02432=1174.650,77.574,-50.282,-179.217,6.130,148.872
C02433=1174.655,77.324,-50.264,-179.219,6.129,148.872
C02434=1174.660,77.075,-50.248,-179.222,6.128,148.873
C02435=1174.665,76.825,-50.231,-179.224,6.127,148.873
C02436=1174.670,76.576,-50.213,-179.227,6.125,148.874
C02437=1174.675,76.326,-50.196,-179.229,6.124,148.874
C02438=1174.680,76.077,-50.179,-179.233,6.123,148.875
C02439=1174.684,75.828,-50.161,-179.235,6.122,148.875
C02440=1174.690,75.579,-50.145,-179.238,6.121,148.876
C02441=1174.694,75.329,-50.128,-179.240,6.120,148.876
C02442=1174.700,75.079,-50.111,-179.243,6.119,148.877
C02443=1174.704,74.830,-50.094,-179.246,6.118,148.877
C02444=1174.709,74.581,-50.076,-179.248,6.117,148.878
C02445=1174.714,74.332,-50.060,-179.251,6.116,148.879
C02446=1174.719,74.082,-50.042,-179.253,6.115,148.879
C02447=1174.724,73.833,-50.026,-179.256,6.113,148.880
C02448=1174.729,73.583,-50.008,-179.258,6.112,148.880
C02449=1174.734,73.335,-49.991,-179.262,6.111,148.881
C02450=1174.739,73.085,-49.974,-179.264,6.110,148.881
C02451=1174.744,72.835,-49.957,-179.267,6.109,148.882
C02452=1174.749,72.586,-49.940,-179.269,6.108,148.882
C02453=1174.754,72.337,-49.924,-179.272,6.108,148.883
C02454=1174.759,72.087,-49.907,-179.274,6.106,148.883
C02455=1174.764,71.838,-49.890,-179.277,6.105,148.884
C02456=1174.769,71.588,-49.873,-179.280,6.104,148.884
C02457=1174.774,71.340,-49.856,-179.282,6.103,148.885
C02458=1174.778,71.090,-49.839,-179.285,6.101,148.885
C02459=1174.783,70.840,-49.822,-179.288,6.101,148.886
C02460=1174.788,70.591,-49.805,-179.290,6.100,148.887
C02461=1174.794,70.342,-49.788,-179.293,6.099,148.887
C02462=1174.798,70.092,-49.772,-179.295,6.098,148.888
C02463=1174.802,69.843,-49.755,-179.299,6.096,148.888
C02464=1174.808,69.594,-49.738,-179.301,6.096,148.889
C02465=1174.813,69.344,-49.721,-179.303,6.095,148.889
C02466=1174.818,69.094,-49.704,-179.306,6.093,148.890
C02467=1174.822,68.845,-49.687,-179.309,6.093,148.890
C02468=1174.828,68.596,-49.671,-179.311,6.091,148.891
C02469=1174.833,68.346,-49.654,-179.314,6.091,148.892
C02470=1174.837,68.097,-49.637,-179.317,6.089,148.892
C02471=1174.842,67.848,-49.621,-179.319,6.088,148.893
C02472=1174.848,67.598,-49.604,-179.322,6.087,148.893
C02473=1174.852,67.349,-49.587,-179.325,6.086,148.894
C02474=1174.857,67.100,-49.571,-179.327,6.085,148.894
C02475=1174.862,66.850,-49.553,-179.330,6.084,148.895
C02476=1174.867,66.600,-49.537,-179.332,6.083,148.895
C02477=1174.872,66.351,-49.521,-179.335,6.083,148.896
C02478=1174.877,66.102,-49.504,-179.338,6.081,148.896
C02479=1174.882,65.852,-49.487,-179.340,6.080,148.897
C02480=1174.887,65.603,-49.471,-179.342,6.079,148.897
C02481=1174.891,65.354,-49.454,-179.346,6.078,148.898
C02482=1174.897,65.104,-49.437,-179.348,6.077,148.899
C02483=1174.902,64.855,-49.421,-179.351,6.076,148.899
C02484=1174.907,64.605,-49.405,-179.353,6.075,148.900
C02485=1174.912,64.356,-49.388,-179.356,6.075,148.900
C02486=1174.917,64.107,-49.371,-179.359,6.073,148.901
C02487=1174.921,63.857,-49.354,-179.361,6.072,148.901
C02488=1174.926,63.608,-49.338,-179.364,6.071,148.902
C02489=1174.931,63.358,-49.322,-179.367,6.070,148.902
C02490=1174.937,63.109,-49.305,-179.369,6.069,148.903
C02491=1174.941,62.860,-49.289,-179.372,6.068,148.904
C02492=1174.946,62.610,-49.272,-179.374,6.067,148.904
C02493=1174.951,62.361,-49.256,-179.377,6.066,148.905
C02494=1174.956,62.111,-49.240,-179.379,6.065,148.905
C02495=1174.961,61.863,-49.223,-179.382,6.064,148.906
C02496=1174.966,61.613,-49.206,-179.385,6.063,148.906
C02497=1174.972,61.363,-49.190,-179.387,6.062,148.907
C02498=1174.976,61.114,-49.174,-179.390,6.061,148.907
C02499=1174.980,60.864,-49.157,-179.393,6.060,148.908
C02500=1174.986,60.615,-49.142,-179.395,6.059,148.908
C02501=1174.990,60.365,-49.125,-179.398,6.058,148.909
C02502=1174.996,60.116,-49.108,-179.400,6.057,148.910
C02503=1175.001,59.866,-49.092,-179.403,6.056,148.910
C02504=1175.006,59.617,-49.076,-179.405,6.055,148.911
C02505=1175.011,59.368,-49.059,-179.408,6.054,148.911
C02506=1175.016,59.119,-49.043,-179.411,6.054,148.912
C02507=1175.020,58.869,-49.027,-179.413,6.053,148.912
C02508=1175.025,58.620,-49.011,-179.416,6.051,148.913
C02509=1175.030,58.370,-48.995,-179.418,6.050,148.913
C02510=1175.036,58.121,-48.978,-179.421,6.050,148.914
C02511=1175.041,57.871,-48.962,-179.424,6.048,148.915
C02512=1175.046,57.622,-48.945,-179.426,6.048,148.915
C02513=1175.051,57.372,-48.929,-179.429,6.047,148.916
C02514=1175.056,57.123,-48.913,-179.432,6.046,148.916
C02515=1175.060,56.874,-48.896,-179.434,6.045,148.917
C02516=1175.066,56.624,-48.881,-179.437,6.044,148.917
C02517=1175.070,56.375,-48.864,-179.439,6.042,148.918
C02518=1175.076,56.126,-48.849,-179.442,6.042,148.919
C02519=1175.080,55.876,-48.832,-179.444,6.041,148.919
C02520=1175.085,55.627,-48.816,-179.447,6.040,148.920
C02521=1175.090,55.377,-48.800,-179.450,6.039,148.920
C02522=1175.095,55.128,-48.784,-179.452,6.038,148.921
C02523=1175.100,54.878,-48.767,-179.455,6.037,148.921
C02524=1175.105,54.610,-48.750,-179.458,6.036,148.922
C02525=1175.111,54.341,-48.733,-179.461,6.035,148.923
C02526=1175.116,54.073,-48.716,-179.463,6.034,148.923
C02527=1175.121,53.804,-48.699,-179.467,6.033,148.924
C02528=1175.126,53.555,-48.683,-179.469,6.032,148.924
C02529=1175.131,53.305,-48.667,-179.471,6.032,148.925
C02530=1175.136,53.056,-48.650,-179.474,6.030,148.925
C02531=1175.142,52.807,-48.635,-179.477,6.029,148.926
C02532=1175.146,52.557,-48.619,-179.479,6.029,148.927
C02533=1175.152,52.308,-48.603,-179.482,6.027,148.927
C02534=1175.156,52.058,-48.587,-179.484,6.026,148.928
C02535=1175.161,51.809,-48.570,-179.487,6.026,148.928
C02536=1175.167,51.559,-48.555,-179.490,6.025,148.929
C02537=1175.172,51.309,-48.539,-179.492,6.024,148.929
C02538=1175.177,51.061,-48.522,-179.495,6.023,148.930
C02539=1175.181,50.811,-48.507,-179.497,6.022,148.931
C02540=1175.186,50.561,-48.492,-179.500,6.021,148.931
C02541=1175.192,50.312,-48.476,-179.503,6.020,148.932
C02542=1175.196,50.062,-48.459,-179.505,6.020,148.932
C02543=1175.201,49.813,-48.444,-179.508,6.018,148.933
C02544=1175.207,49.564,-48.428,-179.511,6.017,148.933
C02545=1175.211,49.314,-48.411,-179.513,6.017,148.934
C02546=1175.217,49.065,-48.396,-179.515,6.016,148.935
C02547=1175.221,48.815,-48.380,-179.519,6.015,148.935
C02548=1175.226,48.566,-48.365,-179.521,6.014,148.936
C02549=1175.231,48.317,-48.349,-179.523,6.013,148.936
C02550=1175.236,48.067,-48.333,-179.526,6.012,148.937
C02551=1175.241,47.817,-48.317,-179.529,6.011,148.937
C02552=1175.247,47.568,-48.301,-179.531,6.011,148.938
C02553=1175.251,47.318,-48.286,-179.534,6.010,148.939
C02554=1175.256,47.069,-48.270,-179.537,6.009,148.939
C02555=1175.261,46.820,-48.254,-179.539,6.008,148.940
C02556=1175.266,46.570,-48.238,-179.542,6.007,148.940
C02557=1175.271,46.320,-48.223,-179.544,6.005,148.941
C02558=1175.276,46.071,-48.208,-179.547,6.005,148.941
C02559=1175.281,45.821,-48.192,-179.550,6.004,148.942
C02560=1175.286,45.572,-48.176,-179.552,6.004,148.943
C02561=1175.291,45.323,-48.160,-179.555,6.002,148.943
C02562=1175.296,45.074,-48.145,-179.557,6.001,148.944
C02563=1175.301,44.824,-48.129,-179.560,6.001,148.944
C02564=1175.306,44.574,-48.113,-179.562,6.000,148.945
C02565=1175.312,44.325,-48.098,-179.565,5.999,148.945
C02566=1175.316,44.075,-48.082,-179.568,5.998,148.946
C02567=1175.321,43.826,-48.067,-179.570,5.997,148.947
C02568=1175.326,43.576,-48.051,-179.573,5.997,148.947
C02569=1175.331,43.327,-48.036,-179.575,5.995,148.948
C02570=1175.336,43.077,-48.020,-179.578,5.995,148.948
C02571=1175.341,42.828,-48.005,-179.580,5.994,148.949
C02572=1175.347,42.578,-47.989,-179.583,5.993,148.949
C02573=1175.351,42.329,-47.974,-179.586,5.992,148.950
C02574=1175.356,42.079,-47.958,-179.588,5.991,148.951
C02575=1175.361,41.830,-47.943,-179.591,5.991,148.951
C02576=1175.366,41.581,-47.928,-179.593,5.990,148.952
C02577=1175.371,41.331,-47.912,-179.596,5.989,148.952
C02578=1175.377,41.082,-47.896,-179.599,5.988,148.953
C02579=1175.381,40.832,-47.881,-179.601,5.987,148.953
C02580=1175.386,40.583,-47.865,-179.604,5.987,148.954
C02581=1175.392,40.333,-47.850,-179.606,5.985,148.955
C02582=1175.396,40.084,-47.835,-179.609,5.984,148.955
C02583=1175.401,39.834,-47.819,-179.611,5.984,148.956
C02584=1175.406,39.585,-47.804,-179.614,5.983,148.956
C02585=1175.411,39.336,-47.788,-179.616,5.983,148.957
C02586=1175.416,39.086,-47.773,-179.619,5.981,148.957
C02587=1175.421,38.837,-47.758,-179.622,5.980,148.958
C02588=1175.427,38.587,-47.743,-179.624,5.980,148.959
C02589=1175.431,38.337,-47.727,-179.627,5.979,148.959
C02590=1175.436,38.088,-47.712,-179.630,5.978,148.960
C02591=1175.442,37.839,-47.696,-179.632,5.977,148.960
C02592=1175.446,37.589,-47.681,-179.635,5.976,148.961
C02593=1175.452,37.340,-47.666,-179.637,5.976,148.962
C02594=1175.457,37.090,-47.651,-179.639,5.975,148.962
C02595=1175.461,36.840,-47.636,-179.643,5.974,148.963
C02596=1175.466,36.591,-47.621,-179.645,5.973,148.963
C02597=1175.471,36.342,-47.605,-179.647,5.972,148.964
C02598=1175.476,36.093,-47.590,-179.650,5.972,148.964
C02599=1175.482,35.843,-47.575,-179.653,5.970,148.965
C02600=1175.486,35.594,-47.560,-179.655,5.970,148.966
C02601=1175.492,35.344,-47.544,-179.658,5.969,148.966
C02602=1175.496,35.094,-47.529,-179.660,5.968,148.967
C02603=1175.502,34.844,-47.514,-179.662,5.968,148.967
C02604=1175.506,34.595,-47.499,-179.666,5.966,148.968
C02605=1175.512,34.346,-47.484,-179.668,5.966,148.969
C02606=1175.516,34.097,-47.469,-179.670,5.965,148.969
C02607=1175.522,33.847,-47.454,-179.673,5.964,148.970
C02608=1175.527,33.598,-47.439,-179.675,5.964,148.970
C02609=1175.532,33.348,-47.423,-179.678,5.962,148.971
C02610=1175.537,33.099,-47.409,-179.681,5.962,148.972
C02611=1175.542,32.849,-47.393,-179.683,5.961,148.972
C02612=1175.546,32.599,-47.378,-179.686,5.960,148.973
C02613=1175.552,32.349,-47.363,-179.688,5.959,148.973
C02614=1175.557,32.100,-47.348,-179.691,5.959,148.974
C02615=1175.561,31.851,-47.333,-179.694,5.958,148.975
C02616=1175.567,31.601,-47.318,-179.696,5.957,148.975
C02617=1175.572,31.352,-47.303,-179.699,5.956,148.976
C02618=1175.577,31.103,-47.288,-179.701,5.956,148.976
C02619=1175.582,30.853,-47.273,-179.704,5.955,148.977
C02620=1175.587,30.604,-47.258,-179.707,5.954,148.977
C02621=1175.592,30.354,-47.244,-179.709,5.953,148.978
C02622=1175.597,30.105,-47.229,-179.712,5.952,148.979
C02623=1175.602,29.855,-47.213,-179.714,5.952,148.979
C02624=1175.607,29.606,-47.199,-179.716,5.951,148.980
C02625=1175.612,29.356,-47.184,-179.719,5.951,148.980
C02626=1175.618,29.106,-47.169,-179.722,5.949,148.981
C02627=1175.622,28.857,-47.154,-179.724,5.948,148.982
C02628=1175.627,28.589,-47.138,-179.727,5.948,148.982
C02629=1175.633,28.319,-47.122,-179.730,5.947,148.983
C02630=1175.638,28.051,-47.106,-179.733,5.946,148.983
C02631=1175.644,27.782,-47.090,-179.735,5.945,148.984
C02632=1175.649,27.532,-47.076,-179.738,5.945,148.985
C02633=1175.654,27.283,-47.061,-179.740,5.944,148.985
C02634=1175.660,27.033,-47.046,-179.743,5.943,148.986
C02635=1175.664,26.784,-47.031,-179.746,5.942,148.987
C02636=1175.669,26.534,-47.016,-179.748,5.941,148.987
C02637=1175.675,26.285,-47.001,-179.751,5.941,148.988
C02638=1175.680,26.035,-46.987,-179.753,5.940,148.988
C02639=1175.684,25.786,-46.972,-179.755,5.939,148.989
C02640=1175.689,25.536,-46.957,-179.758,5.939,148.989
C02641=1175.695,25.286,-46.942,-179.761,5.938,148.990
C02642=1175.700,25.037,-46.927,-179.764,5.937,148.991
C02643=1175.704,24.787,-46.913,-179.766,5.936,148.991
C02644=1175.709,24.538,-46.898,-179.768,5.935,148.992
C02645=1175.715,24.288,-46.883,-179.771,5.935,148.992
C02646=1175.720,24.038,-46.869,-179.774,5.934,148.993
C02647=1175.724,23.789,-46.854,-179.776,5.934,148.994
C02648=1175.729,23.540,-46.840,-179.779,5.932,148.994
C02649=1175.734,23.290,-46.825,-179.782,5.932,148.995
C02650=1175.740,23.040,-46.810,-179.784,5.931,148.995
C02651=1175.745,22.791,-46.796,-179.786,5.931,148.996
C02652=1175.750,22.542,-46.782,-179.789,5.930,148.996
C02653=1175.755,22.293,-46.767,-179.791,5.929,148.997
C02654=1175.760,22.043,-46.752,-179.794,5.929,148.998
C02655=1175.766,21.793,-46.738,-179.797,5.927,148.998
C02656=1175.770,21.544,-46.723,-179.799,5.927,148.999
C02657=1175.775,21.294,-46.708,-179.802,5.926,149.000
C02658=1175.780,21.044,-46.694,-179.804,5.925,149.000
C02659=1175.785,20.795,-46.680,-179.807,5.925,149.001
C02660=1175.790,20.546,-46.665,-179.809,5.924,149.001
C02661=1175.795,20.296,-46.650,-179.812,5.923,149.002
C02662=1175.801,20.047,-46.636,-179.814,5.923,149.003
C02663=1175.806,19.797,-46.622,-179.816,5.922,149.003
C02664=1175.811,19.547,-46.607,-179.820,5.921,149.004
C02665=1175.815,19.298,-46.592,-179.822,5.920,149.004
C02666=1175.820,19.048,-46.578,-179.824,5.919,149.005
C02667=1175.825,18.799,-46.564,-179.827,5.919,149.006
C02668=1175.830,18.549,-46.550,-179.830,5.918,149.006
C02669=1175.836,18.300,-46.536,-179.832,5.918,149.007
C02670=1175.841,18.051,-46.520,-179.835,5.917,149.007
C02671=1175.846,17.801,-46.506,-179.837,5.916,149.008
C02672=1175.851,17.551,-46.491,-179.839,5.916,149.009
C02673=1175.856,17.301,-46.477,-179.843,5.915,149.009
C02674=1175.861,17.052,-46.463,-179.845,5.914,149.010
C02675=1175.867,16.803,-46.449,-179.847,5.913,149.010
C02676=1175.872,16.553,-46.435,-179.850,5.913,149.011
C02677=1175.877,16.303,-46.420,-179.852,5.912,149.011
C02678=1175.882,16.054,-46.406,-179.855,5.911,149.012
C02679=1175.886,15.804,-46.391,-179.858,5.911,149.013
C02680=1175.891,15.555,-46.377,-179.860,5.910,149.013
C02681=1175.897,15.306,-46.363,-179.862,5.910,149.014
C02682=1175.902,15.056,-46.349,-179.865,5.909,149.014
C02683=1175.907,14.806,-46.334,-179.867,5.908,149.015
C02684=1175.912,14.557,-46.320,-179.870,5.907,149.016
C02685=1175.917,14.307,-46.306,-179.873,5.906,149.016
C02686=1175.922,14.058,-46.292,-179.875,5.906,149.017
C02687=1175.927,13.808,-46.278,-179.878,5.905,149.018
C02688=1175.932,13.558,-46.263,-179.880,5.904,149.018
C02689=1175.937,13.309,-46.249,-179.883,5.904,149.019
C02690=1175.942,13.060,-46.235,-179.885,5.903,149.019
C02691=1175.947,12.810,-46.221,-179.888,5.903,149.020
C02692=1175.952,12.560,-46.207,-179.890,5.902,149.021
C02693=1175.957,12.311,-46.192,-179.893,5.902,149.021
C02694=1175.963,12.062,-46.179,-179.895,5.901,149.022
C02695=1175.968,11.812,-46.164,-179.898,5.900,149.022
C02696=1175.973,11.562,-46.150,-179.900,5.899,149.023
C02697=1175.978,11.312,-46.136,-179.903,5.898,149.024
C02698=1175.983,11.063,-46.123,-179.906,5.898,149.024
C02699=1175.988,10.813,-46.109,-179.908,5.897,149.025
C02700=1175.993,10.564,-46.095,-179.911,5.896,149.025
C02701=1175.998,10.314,-46.080,-179.913,5.896,149.026
C02702=1176.003,10.065,-46.066,-179.915,5.895,149.027
C02703=1176.008,9.815,-46.052,-179.918,5.895,149.027
C02704=1176.013,9.566,-46.038,-179.921,5.894,149.028
C02705=1176.018,9.316,-46.023,-179.923,5.893,149.028
C02706=1176.024,9.066,-46.010,-179.925,5.893,149.029
C02707=1176.028,8.817,-45.997,-179.928,5.892,149.030
C02708=1176.033,8.567,-45.982,-179.930,5.891,149.030
C02709=1176.039,8.318,-45.968,-179.933,5.891,149.031
C02710=1176.044,8.068,-45.954,-179.936,5.891,149.032
C02711=1176.049,7.819,-45.940,-179.938,5.890,149.032
C02712=1176.055,7.569,-45.927,-179.940,5.889,149.033
C02713=1176.060,7.319,-45.912,-179.943,5.889,149.033
C02714=1176.064,7.070,-45.899,-179.946,5.887,149.034
C02715=1176.069,6.821,-45.885,-179.948,5.887,149.035
C02716=1176.074,6.571,-45.871,-179.951,5.886,149.035
C02717=1176.079,6.321,-45.857,-179.953,5.885,149.036
C02718=1176.085,6.072,-45.843,-179.956,5.885,149.036
C02719=1176.089,5.823,-45.829,-179.958,5.884,149.037
C02720=1176.094,5.573,-45.815,-179.961,5.884,149.038
C02721=1176.100,5.323,-45.802,-179.963,5.883,149.038
C02722=1176.105,5.073,-45.788,-179.966,5.882,149.039
C02723=1176.109,4.824,-45.774,-179.968,5.882,149.039
C02724=1176.115,4.574,-45.761,-179.971,5.881,149.040
C02725=1176.120,4.325,-45.746,-179.973,5.880,149.040
C02726=1176.125,4.075,-45.732,-179.976,5.880,149.041
C02727=1176.130,3.826,-45.720,-179.978,5.879,149.042
C02728=1176.135,3.576,-45.705,-179.981,5.879,149.042
C02729=1176.141,3.327,-45.691,-179.983,5.878,149.043
C02730=1176.146,3.077,-45.678,-179.986,5.878,149.044
C02731=1176.150,2.827,-45.664,-179.988,5.877,149.044
C02732=1176.156,2.559,-45.650,-179.991,5.876,149.045
C02733=1176.162,2.289,-45.635,-179.993,5.876,149.046
C02734=1176.167,2.020,-45.620,-179.997,5.875,149.046
C02735=1176.172,1.750,-45.605,-179.999,5.874,149.047
C02736=1176.178,1.501,-45.591,179.999,5.873,149.047
C02737=1176.183,1.251,-45.578,179.996,5.873,149.048
C02738=1176.188,1.002,-45.564,179.993,5.872,149.049
C02739=1176.193,0.752,-45.550,179.991,5.872,149.049
C02740=1176.198,0.503,-45.537,179.988,5.871,149.050
C02741=1176.203,0.253,-45.523,179.986,5.871,149.051
C02742=1176.208,0.003,-45.509,179.984,5.870,149.051
C02743=1176.214,-0.246,-45.496,179.981,5.869,149.052
C02744=1176.218,-0.496,-45.482,179.978,5.869,149.052
C02745=1176.224,-0.745,-45.469,179.976,5.868,149.053
C02746=1176.229,-0.995,-45.455,179.974,5.868,149.054
C02747=1176.234,-1.244,-45.442,179.971,5.867,149.054
C02748=1176.239,-1.494,-45.428,179.969,5.866,149.055
C02749=1176.244,-1.744,-45.415,179.966,5.866,149.055
C02750=1176.249,-1.993,-45.401,179.963,5.865,149.056
C02751=1176.254,-2.243,-45.388,179.961,5.865,149.057
C02752=1176.260,-2.492,-45.374,179.959,5.864,149.057
C02753=1176.264,-2.742,-45.361,179.956,5.864,149.058
C02754=1176.270,-2.991,-45.347,179.954,5.863,149.058
C02755=1176.275,-3.242,-45.334,179.951,5.862,149.059
C02756=1176.280,-3.490,-45.320,179.948,5.862,149.060
C02757=1176.285,-3.741,-45.307,179.946,5.861,149.060
C02758=1176.290,-3.990,-45.294,179.944,5.861,149.061
C02759=1176.295,-4.240,-45.280,179.941,5.860,149.062
C02760=1176.300,-4.489,-45.267,179.939,5.859,149.062
C02761=1176.305,-4.739,-45.253,179.936,5.859,149.063
C02762=1176.311,-4.988,-45.240,179.933,5.858,149.063
C02763=1176.315,-5.238,-45.227,179.931,5.857,149.064
C02764=1176.321,-5.487,-45.213,179.929,5.857,149.065
C02765=1176.326,-5.737,-45.200,179.926,5.857,149.065
C02766=1176.331,-5.987,-45.187,179.924,5.856,149.066
C02767=1176.336,-6.236,-45.173,179.921,5.855,149.066
C02768=1176.342,-6.486,-45.160,179.919,5.855,149.067
C02769=1176.347,-6.735,-45.147,179.916,5.854,149.068
C02770=1176.352,-6.985,-45.133,179.914,5.854,149.068
C02771=1176.357,-7.234,-45.120,179.912,5.854,149.069
C02772=1176.362,-7.485,-45.107,179.909,5.853,149.069
C02773=1176.367,-7.733,-45.094,179.907,5.853,149.070
C02774=1176.372,-7.984,-45.080,179.904,5.852,149.071
C02775=1176.377,-8.233,-45.067,179.902,5.851,149.071
C02776=1176.382,-8.483,-45.054,179.899,5.851,149.072
C02777=1176.387,-8.732,-45.040,179.897,5.850,149.073
C02778=1176.392,-8.981,-45.028,179.894,5.849,149.073
C02779=1176.398,-9.232,-45.014,179.892,5.849,149.074
C02780=1176.402,-9.480,-45.001,179.889,5.849,149.075
C02781=1176.408,-9.731,-44.987,179.887,5.848,149.075
C02782=1176.413,-9.980,-44.975,179.884,5.847,149.076
C02783=1176.417,-10.230,-44.962,179.882,5.847,149.076
C02784=1176.423,-10.480,-44.949,179.879,5.846,149.077
C02785=1176.428,-10.728,-44.935,179.877,5.846,149.078
C02786=1176.433,-10.979,-44.922,179.874,5.845,149.078
C02787=1176.438,-11.228,-44.909,179.872,5.844,149.079
C02788=1176.443,-11.478,-44.896,179.869,5.844,149.079
C02789=1176.449,-11.728,-44.883,179.867,5.843,149.080
C02790=1176.454,-11.977,-44.870,179.865,5.843,149.081
C02791=1176.459,-12.227,-44.856,179.862,5.842,149.081
C02792=1176.464,-12.476,-44.844,179.859,5.842,149.082
C02793=1176.469,-12.725,-44.831,179.858,5.842,149.082
C02794=1176.474,-12.976,-44.817,179.855,5.841,149.083
C02795=1176.480,-13.225,-44.805,179.852,5.841,149.084
C02796=1176.484,-13.475,-44.792,179.850,5.840,149.084
C02797=1176.490,-13.725,-44.779,179.847,5.839,149.085
C02798=1176.495,-13.974,-44.766,179.845,5.839,149.086
C02799=1176.499,-14.223,-44.752,179.843,5.838,149.086
C02800=1176.505,-14.473,-44.739,179.840,5.838,149.087
C02801=1176.510,-14.722,-44.727,179.837,5.837,149.088
C02802=1176.515,-14.972,-44.714,179.835,5.836,149.088
C02803=1176.521,-15.222,-44.700,179.832,5.836,149.089
C02804=1176.526,-15.471,-44.688,179.830,5.835,149.089
C02805=1176.530,-15.721,-44.675,179.828,5.835,149.090
C02806=1176.535,-15.971,-44.662,179.825,5.834,149.091
C02807=1176.541,-16.220,-44.649,179.823,5.835,149.091
C02808=1176.546,-16.470,-44.636,179.821,5.834,149.092
C02809=1176.551,-16.720,-44.623,179.818,5.833,149.092
C02810=1176.557,-16.969,-44.610,179.815,5.833,149.093
C02811=1176.562,-17.219,-44.598,179.813,5.832,149.094
C02812=1176.566,-17.469,-44.585,179.811,5.831,149.094
C02813=1176.572,-17.718,-44.572,179.808,5.831,149.095
C02814=1176.577,-17.968,-44.559,179.806,5.830,149.095
C02815=1176.582,-18.218,-44.546,179.803,5.830,149.096
C02816=1176.587,-18.467,-44.533,179.800,5.829,149.097
C02817=1176.592,-18.716,-44.521,179.798,5.828,149.097
C02818=1176.598,-18.966,-44.508,179.796,5.828,149.098
C02819=1176.603,-19.216,-44.495,179.794,5.828,149.099
C02820=1176.608,-19.466,-44.483,179.791,5.828,149.099
C02821=1176.613,-19.715,-44.470,179.789,5.827,149.100
C02822=1176.618,-19.964,-44.457,179.786,5.827,149.101
C02823=1176.623,-20.215,-44.444,179.784,5.826,149.101
C02824=1176.629,-20.464,-44.431,179.781,5.825,149.102
C02825=1176.634,-20.713,-44.419,179.779,5.825,149.102
C02826=1176.639,-20.963,-44.406,179.776,5.824,149.103
C02827=1176.643,-21.213,-44.393,179.774,5.824,149.104
C02828=1176.649,-21.463,-44.381,179.771,5.823,149.104
C02829=1176.655,-21.712,-44.368,179.769,5.823,149.105
C02830=1176.660,-21.962,-44.355,179.767,5.823,149.105
C02831=1176.664,-22.212,-44.343,179.764,5.822,149.106
C02832=1176.669,-22.461,-44.330,179.762,5.821,149.107
C02833=1176.675,-22.710,-44.317,179.759,5.821,149.107
C02834=1176.680,-22.960,-44.305,179.757,5.821,149.108
C02835=1176.686,-23.210,-44.292,179.754,5.820,149.108
C02836=1176.691,-23.480,-44.279,179.752,5.819,149.109
C02837=1176.696,-23.749,-44.265,179.749,5.819,149.110
C02838=1176.703,-24.019,-44.252,179.746,5.818,149.110
C02839=1176.708,-24.289,-44.238,179.744,5.818,149.111
C02840=1176.713,-24.538,-44.225,179.741,5.818,149.112
C02841=1176.718,-24.788,-44.213,179.739,5.817,149.112
C02842=1176.723,-25.038,-44.201,179.736,5.816,149.113
C02843=1176.728,-25.288,-44.188,179.734,5.817,149.114
C02844=1176.733,-25.537,-44.175,179.732,5.816,149.114
C02845=1176.738,-25.786,-44.163,179.729,5.815,149.115
C02846=1176.744,-26.036,-44.150,179.727,5.815,149.116
C02847=1176.749,-26.286,-44.137,179.725,5.814,149.116
C02848=1176.754,-26.536,-44.125,179.722,5.814,149.117
C02849=1176.759,-26.786,-44.113,179.719,5.813,149.117
C02850=1176.764,-27.035,-44.100,179.717,5.812,149.118
C02851=1176.769,-27.284,-44.088,179.715,5.813,149.119
C02852=1176.775,-27.534,-44.076,179.712,5.812,149.119
C02853=1176.780,-27.784,-44.063,179.710,5.811,149.120
C02854=1176.785,-28.034,-44.050,179.708,5.811,149.121
C02855=1176.790,-28.284,-44.038,179.705,5.811,149.121
C02856=1176.795,-28.533,-44.026,179.703,5.810,149.122
C02857=1176.800,-28.782,-44.013,179.700,5.809,149.122
C02858=1176.806,-29.032,-44.001,179.698,5.810,149.123
C02859=1176.811,-29.281,-43.989,179.696,5.809,149.124
C02860=1176.816,-29.531,-43.977,179.693,5.808,149.124
C02861=1176.821,-29.781,-43.964,179.690,5.808,149.125
C02862=1176.826,-30.031,-43.951,179.688,5.807,149.125
C02863=1176.831,-30.281,-43.939,179.686,5.807,149.126
C02864=1176.836,-30.530,-43.927,179.683,5.806,149.127
C02865=1176.842,-30.780,-43.915,179.681,5.806,149.127
C02866=1176.847,-31.029,-43.902,179.679,5.806,149.128
C02867=1176.852,-31.279,-43.891,179.676,5.805,149.129
C02868=1176.857,-31.528,-43.878,179.674,5.805,149.129
C02869=1176.862,-31.777,-43.866,179.671,5.804,149.130
C02870=1176.867,-32.027,-43.854,179.669,5.804,149.131
C02871=1176.872,-32.277,-43.841,179.666,5.803,149.131
C02872=1176.878,-32.527,-43.829,179.664,5.803,149.132
C02873=1176.882,-32.777,-43.816,179.662,5.803,149.132
C02874=1176.888,-33.027,-43.804,179.659,5.802,149.133
C02875=1176.893,-33.276,-43.792,179.657,5.802,149.134
C02876=1176.898,-33.526,-43.780,179.654,5.801,149.134
C02877=1176.904,-33.776,-43.768,179.652,5.800,149.135
C02878=1176.909,-34.025,-43.755,179.650,5.801,149.135
C02879=1176.914,-34.275,-43.744,179.647,5.800,149.136
C02880=1176.919,-34.524,-43.732,179.645,5.799,149.137
C02881=1176.924,-34.774,-43.720,179.642,5.799,149.137
C02882=1176.929,-35.023,-43.707,179.640,5.798,149.138
C02883=1176.935,-35.273,-43.695,179.637,5.798,149.138
C02884=1176.940,-35.523,-43.683,179.635,5.798,149.139
C02885=1176.945,-35.773,-43.671,179.633,5.797,149.140
C02886=1176.950,-36.022,-43.659,179.631,5.797,149.140
C02887=1176.955,-36.271,-43.647,179.628,5.796,149.141
C02888=1176.961,-36.521,-43.635,179.626,5.796,149.142
C02889=1176.966,-36.771,-43.622,179.624,5.796,149.142
C02890=1176.971,-37.021,-43.610,179.621,5.795,149.143
C02891=1176.976,-37.271,-43.599,179.619,5.795,149.143
C02892=1176.981,-37.520,-43.587,179.616,5.794,149.144
C02893=1176.986,-37.770,-43.575,179.613,5.794,149.145
C02894=1176.992,-38.019,-43.563,179.611,5.793,149.145
C02895=1176.997,-38.269,-43.550,179.609,5.793,149.146
C02896=1177.002,-38.519,-43.538,179.607,5.793,149.147
C02897=1177.007,-38.768,-43.527,179.604,5.792,149.147
C02898=1177.012,-39.018,-43.514,179.602,5.792,149.148
C02899=1177.018,-39.268,-43.503,179.599,5.791,149.149
C02900=1177.023,-39.518,-43.491,179.597,5.791,149.149
C02901=1177.028,-39.767,-43.479,179.595,5.791,149.150
C02902=1177.033,-40.016,-43.467,179.592,5.790,149.150
C02903=1177.038,-40.266,-43.455,179.590,5.789,149.151
C02904=1177.044,-40.516,-43.443,179.587,5.789,149.152
C02905=1177.048,-40.766,-43.432,179.585,5.789,149.152
C02906=1177.053,-41.015,-43.419,179.583,5.789,149.153
C02907=1177.059,-41.265,-43.407,179.580,5.788,149.153
C02908=1177.065,-41.514,-43.396,179.578,5.788,149.154
C02909=1177.070,-41.764,-43.384,179.576,5.787,149.155
C02910=1177.075,-42.013,-43.372,179.573,5.787,149.155
C02911=1177.080,-42.263,-43.360,179.571,5.787,149.156
C02912=1177.085,-42.513,-43.349,179.569,5.786,149.157
C02913=1177.090,-42.763,-43.337,179.566,5.786,149.157
C02914=1177.096,-43.013,-43.325,179.563,5.785,149.158
C02915=1177.101,-43.262,-43.312,179.562,5.785,149.158
C02916=1177.106,-43.512,-43.301,179.559,5.785,149.159
C02917=1177.111,-43.762,-43.289,179.556,5.784,149.160
C02918=1177.116,-44.012,-43.277,179.554,5.784,149.160
C02919=1177.121,-44.261,-43.266,179.552,5.783,149.161
C02920=1177.127,-44.511,-43.254,179.550,5.783,149.161
C02921=1177.132,-44.760,-43.242,179.547,5.783,149.162
C02922=1177.137,-45.009,-43.230,179.545,5.782,149.163
C02923=1177.142,-45.259,-43.219,179.542,5.781,149.163
C02924=1177.147,-45.509,-43.207,179.540,5.781,149.164
C02925=1177.152,-45.759,-43.195,179.538,5.781,149.165
C02926=1177.158,-46.009,-43.184,179.535,5.781,149.165
C02927=1177.163,-46.259,-43.172,179.533,5.780,149.166
C02928=1177.168,-46.508,-43.160,179.530,5.780,149.167
C02929=1177.174,-46.758,-43.149,179.529,5.780,149.167
C02930=1177.179,-47.007,-43.138,179.526,5.779,149.168
C02931=1177.184,-47.257,-43.126,179.523,5.779,149.168
C02932=1177.189,-47.506,-43.114,179.521,5.778,149.169
C02933=1177.194,-47.756,-43.102,179.518,5.778,149.170
C02934=1177.199,-48.006,-43.090,179.516,5.778,149.170
C02935=1177.204,-48.256,-43.079,179.514,5.777,149.171
C02936=1177.210,-48.505,-43.067,179.511,5.777,149.172
C02937=1177.215,-48.755,-43.056,179.509,5.776,149.172
C02938=1177.220,-49.005,-43.044,179.507,5.776,149.173
C02939=1177.225,-49.254,-43.033,179.505,5.776,149.173
C02940=1177.231,-49.524,-43.021,179.502,5.775,149.174
C02941=1177.236,-49.795,-43.008,179.499,5.775,149.175
C02942=1177.242,-50.066,-42.996,179.497,5.774,149.175
C02943=1177.248,-50.335,-42.983,179.494,5.774,149.176
C02944=1177.253,-50.585,-42.971,179.492,5.773,149.177
C02945=1177.258,-50.835,-42.960,179.490,5.774,149.177
C02946=1177.264,-51.085,-42.948,179.487,5.773,149.178
C02947=1177.268,-51.335,-42.937,179.485,5.772,149.179
C02948=1177.274,-51.584,-42.925,179.482,5.772,149.179
C02949=1177.279,-51.833,-42.914,179.481,5.772,149.180
C02950=1177.285,-52.084,-42.903,179.478,5.772,149.180
C02951=1177.289,-52.334,-42.891,179.476,5.771,149.181
C02952=1177.295,-52.583,-42.880,179.473,5.770,149.182
C02953=1177.300,-52.832,-42.868,179.471,5.771,149.182
C02954=1177.306,-53.082,-42.857,179.469,5.770,149.183
C02955=1177.310,-53.332,-42.845,179.466,5.770,149.184
C02956=1177.316,-53.582,-42.833,179.463,5.769,149.184
C02957=1177.321,-53.831,-42.823,179.462,5.769,149.185
C02958=1177.326,-54.081,-42.811,179.459,5.769,149.185
C02959=1177.331,-54.331,-42.800,179.456,5.768,149.186
C02960=1177.336,-54.581,-42.789,179.455,5.768,149.187
C02961=1177.342,-54.830,-42.777,179.452,5.768,149.187
C02962=1177.347,-55.080,-42.766,179.450,5.767,149.188
C02963=1177.352,-55.329,-42.754,179.447,5.767,149.188
C02964=1177.357,-55.579,-42.743,179.445,5.767,149.189
C02965=1177.363,-55.829,-42.733,179.443,5.766,149.190
C02966=1177.368,-56.079,-42.721,179.440,5.766,149.190
C02967=1177.373,-56.328,-42.709,179.438,5.765,149.191
C02968=1177.378,-56.578,-42.698,179.436,5.765,149.192
C02969=1177.383,-56.827,-42.687,179.433,5.765,149.192
C02970=1177.388,-57.077,-42.676,179.431,5.764,149.193
C02971=1177.394,-57.327,-42.664,179.429,5.764,149.193
C02972=1177.398,-57.577,-42.653,179.427,5.764,149.194
C02973=1177.405,-57.826,-42.641,179.424,5.763,149.195
C02974=1177.410,-58.076,-42.631,179.422,5.763,149.195
C02975=1177.414,-58.326,-42.619,179.420,5.763,149.196
C02976=1177.420,-58.575,-42.608,179.417,5.762,149.197
C02977=1177.425,-58.825,-42.597,179.415,5.762,149.197
C02978=1177.430,-59.075,-42.586,179.412,5.762,149.198
C02979=1177.436,-59.324,-42.575,179.411,5.762,149.198
C02980=1177.441,-59.574,-42.563,179.408,5.761,149.199
C02981=1177.446,-59.824,-42.553,179.406,5.760,149.200
C02982=1177.452,-60.073,-42.541,179.403,5.760,149.200
C02983=1177.456,-60.323,-42.530,179.401,5.760,149.201
C02984=1177.461,-60.573,-42.519,179.399,5.759,149.201
C02985=1177.467,-60.823,-42.508,179.396,5.759,149.202
C02986=1177.472,-61.072,-42.496,179.394,5.759,149.203
C02987=1177.477,-61.322,-42.486,179.392,5.759,149.203
C02988=1177.482,-61.571,-42.475,179.389,5.758,149.204
C02989=1177.488,-61.821,-42.463,179.386,5.758,149.205
C02990=1177.493,-62.072,-42.453,179.385,5.758,149.205
C02991=1177.498,-62.320,-42.442,179.382,5.757,149.206
C02992=1177.504,-62.571,-42.430,179.380,5.757,149.206
C02993=1177.509,-62.821,-42.419,179.378,5.757,149.207
C02994=1177.514,-63.070,-42.408,179.375,5.757,149.208
C02995=1177.519,-63.320,-42.398,179.373,5.756,149.208
C02996=1177.524,-63.570,-42.386,179.371,5.756,149.209
C02997=1177.530,-63.819,-42.376,179.369,5.755,149.210
C02998=1177.535,-64.069,-42.364,179.366,5.755,149.210
C02999=1177.540,-64.318,-42.354,179.363,5.755,149.211
C03000=1177.546,-64.568,-42.342,179.362,5.754,149.211
C03001=1177.550,-64.818,-42.331,179.359,5.754,149.212
C03002=1177.556,-65.068,-42.321,179.357,5.754,149.213
C03003=1177.561,-65.317,-42.309,179.355,5.754,149.213
C03004=1177.566,-65.567,-42.299,179.352,5.753,149.214
C03005=1177.572,-65.817,-42.287,179.350,5.752,149.214
C03006=1177.577,-66.067,-42.277,179.348,5.753,149.215
C03007=1177.582,-66.316,-42.266,179.345,5.752,149.216
C03008=1177.587,-66.566,-42.255,179.343,5.752,149.216
C03009=1177.592,-66.815,-42.244,179.340,5.751,149.217
C03010=1177.598,-67.066,-42.233,179.339,5.751,149.218
C03011=1177.603,-67.315,-42.222,179.336,5.751,149.218
C03012=1177.608,-67.565,-42.212,179.334,5.750,149.219
C03013=1177.613,-67.814,-42.200,179.332,5.750,149.219
C03014=1177.618,-68.064,-42.190,179.329,5.750,149.220
C03015=1177.623,-68.314,-42.180,179.327,5.750,149.221
C03016=1177.629,-68.563,-42.168,179.325,5.750,149.221
C03017=1177.634,-68.814,-42.157,179.322,5.749,149.222
C03018=1177.640,-69.063,-42.147,179.320,5.748,149.223
C03019=1177.645,-69.313,-42.136,179.318,5.749,149.223
C03020=1177.649,-69.562,-42.125,179.315,5.748,149.224
C03021=1177.655,-69.812,-42.114,179.313,5.748,149.224
C03022=1177.660,-70.062,-42.104,179.311,5.748,149.225
C03023=1177.666,-70.311,-42.092,179.309,5.747,149.226
C03024=1177.671,-70.562,-42.082,179.306,5.747,149.226
C03025=1177.677,-70.811,-42.072,179.304,5.747,149.227
C03026=1177.681,-71.061,-42.060,179.302,5.746,149.227
C03027=1177.687,-71.310,-42.050,179.299,5.746,149.228
C03028=1177.692,-71.560,-42.039,179.298,5.746,149.229
C03029=1177.697,-71.810,-42.029,179.295,5.745,149.229
C03030=1177.702,-72.060,-42.018,179.292,5.745,149.230
C03031=1177.708,-72.309,-42.007,179.291,5.745,149.231
C03032=1177.713,-72.559,-41.997,179.288,5.745,149.231
C03033=1177.718,-72.809,-41.986,179.286,5.744,149.232
C03034=1177.724,-73.059,-41.975,179.284,5.744,149.232
C03035=1177.729,-73.308,-41.964,179.281,5.744,149.233
C03036=1177.734,-73.558,-41.954,179.279,5.743,149.234
C03037=1177.740,-73.808,-41.943,179.277,5.743,149.234
C03038=1177.744,-74.057,-41.932,179.275,5.743,149.235
C03039=1177.750,-74.307,-41.922,179.272,5.742,149.236
C03040=1177.755,-74.557,-41.911,179.270,5.743,149.236
C03041=1177.761,-74.807,-41.901,179.268,5.742,149.237
C03042=1177.765,-75.056,-41.890,179.265,5.741,149.237
C03043=1177.771,-75.306,-41.880,179.264,5.741,149.238
C03044=1177.777,-75.578,-41.868,179.261,5.741,149.239
C03045=1177.782,-75.847,-41.857,179.258,5.741,149.239
C03046=1177.788,-76.119,-41.845,179.256,5.740,149.240
C03047=1177.793,-76.390,-41.834,179.253,5.740,149.241
C03048=1177.799,-76.639,-41.823,179.251,5.740,149.241
C03049=1177.804,-76.889,-41.813,179.249,5.739,149.242
C03050=1177.809,-77.139,-41.803,179.247,5.739,149.242
C03051=1177.815,-77.389,-41.792,179.244,5.739,149.243
C03052=1177.820,-77.639,-41.782,179.242,5.739,149.244
C03053=1177.826,-77.888,-41.772,179.240,5.739,149.244
C03054=1177.830,-78.138,-41.760,179.237,5.738,149.245
C03055=1177.836,-78.388,-41.750,179.235,5.737,149.246
C03056=1177.841,-78.637,-41.740,179.233,5.738,149.246
C03057=1177.846,-78.887,-41.729,179.231,5.737,149.247
C03058=1177.852,-79.137,-41.719,179.228,5.737,149.247
C03059=1177.857,-79.387,-41.709,179.226,5.737,149.248
C03060=1177.863,-79.637,-41.698,179.224,5.736,149.249
C03061=1177.868,-79.886,-41.687,179.221,5.736,149.249
C03062=1177.873,-80.136,-41.677,179.220,5.736,149.250
C03063=1177.879,-80.385,-41.667,179.217,5.735,149.251
C03064=1177.883,-80.635,-41.657,179.215,5.735,149.251
C03065=1177.888,-80.885,-41.646,179.213,5.735,149.252
C03066=1177.894,-81.134,-41.636,179.210,5.735,149.252
C03067=1177.899,-81.385,-41.626,179.209,5.735,149.253
C03068=1177.905,-81.634,-41.615,179.206,5.734,149.254
C03069=1177.910,-81.884,-41.605,179.204,5.733,149.254
C03070=1177.915,-82.134,-41.595,179.202,5.734,149.255
C03071=1177.921,-82.384,-41.584,179.199,5.733,149.256
C03072=1177.926,-82.634,-41.574,179.197,5.733,149.256
C03073=1177.931,-82.883,-41.564,179.195,5.733,149.257
C03074=1177.936,-83.133,-41.554,179.192,5.732,149.257
C03075=1177.941,-83.382,-41.543,179.190,5.733,149.258
C03076=1177.947,-83.632,-41.533,179.188,5.732,149.258
C03077=1177.952,-83.881,-41.522,179.186,5.731,149.259
C03078=1177.957,-84.132,-41.512,179.184,5.731,149.260
C03079=1177.962,-84.381,-41.502,179.181,5.731,149.260
C03080=1177.968,-84.630,-41.492,179.179,5.731,149.261
C03081=1177.973,-84.881,-41.482,179.177,5.731,149.261
C03082=1177.978,-85.131,-41.472,179.174,5.730,149.262
C03083=1177.983,-85.381,-41.461,179.173,5.730,149.263
C03084=1177.988,-85.630,-41.452,179.170,5.730,149.263
C03085=1177.994,-85.880,-41.442,179.168,5.729,149.264
C03086=1178.000,-86.129,-41.431,179.166,5.729,149.265
C03087=1178.005,-86.380,-41.421,179.163,5.729,149.265
C03088=1178.010,-86.629,-41.411,179.162,5.729,149.266
C03089=1178.015,-86.878,-41.401,179.159,5.729,149.266
C03090=1178.020,-87.129,-41.390,179.157,5.728,149.267
C03091=1178.026,-87.378,-41.380,179.155,5.728,149.268
C03092=1178.031,-87.628,-41.370,179.152,5.727,149.268
C03093=1178.035,-87.878,-41.360,179.150,5.728,149.269
C03094=1178.041,-88.127,-41.350,179.148,5.727,149.269
C03095=1178.047,-88.377,-41.340,179.145,5.727,149.270
C03096=1178.052,-88.628,-41.330,179.143,5.727,149.271
C03097=1178.057,-88.877,-41.320,179.141,5.726,149.271
C03098=1178.062,-89.126,-41.310,179.139,5.727,149.272
C03099=1178.068,-89.376,-41.300,179.137,5.726,149.272
C03100=1178.073,-89.626,-41.289,179.134,5.726,149.273
C03101=1178.078,-89.875,-41.279,179.133,5.726,149.274
C03102=1178.084,-90.125,-41.270,179.130,5.725,149.274
C03103=1178.089,-90.375,-41.260,179.128,5.725,149.275
C03104=1178.094,-90.625,-41.250,179.126,5.725,149.276
C03105=1178.099,-90.874,-41.240,179.123,5.724,149.276
C03106=1178.105,-91.124,-41.229,179.121,5.724,149.277
C03107=1178.110,-91.374,-41.219,179.119,5.724,149.277
C03108=1178.115,-91.624,-41.210,179.117,5.724,149.278
C03109=1178.121,-91.874,-41.200,179.114,5.724,149.279
C03110=1178.126,-92.123,-41.189,179.112,5.723,149.279
C03111=1178.131,-92.372,-41.180,179.110,5.723,149.280
C03112=1178.136,-92.623,-41.170,179.108,5.722,149.280
C03113=1178.142,-92.873,-41.160,179.106,5.723,149.281
C03114=1178.147,-93.122,-41.150,179.104,5.722,149.281
C03115=1178.152,-93.372,-41.140,179.101,5.722,149.282
C03116=1178.158,-93.622,-41.130,179.099,5.722,149.283
C03117=1178.163,-93.872,-41.120,179.097,5.721,149.283
C03118=1178.168,-94.121,-41.110,179.095,5.721,149.284
C03119=1178.174,-94.371,-41.100,179.093,5.721,149.285
C03120=1178.179,-94.621,-41.091,179.090,5.721,149.285
C03121=1178.184,-94.871,-41.081,179.088,5.720,149.286
C03122=1178.189,-95.120,-41.071,179.086,5.720,149.287
C03123=1178.195,-95.370,-41.061,179.084,5.720,149.287
C03124=1178.200,-95.620,-41.051,179.081,5.720,149.288
C03125=1178.205,-95.869,-41.042,179.080,5.720,149.288
C03126=1178.211,-96.119,-41.032,179.077,5.719,149.289
C03127=1178.215,-96.369,-41.022,179.075,5.719,149.289
C03128=1178.221,-96.619,-41.012,179.073,5.719,149.290
C03129=1178.227,-96.869,-41.002,179.071,5.718,149.291
C03130=1178.232,-97.118,-40.993,179.068,5.719,149.291
C03131=1178.237,-97.368,-40.983,179.066,5.718,149.292
C03132=1178.242,-97.618,-40.974,179.064,5.718,149.292
C03133=1178.247,-97.868,-40.963,179.062,5.717,149.293
C03134=1178.253,-98.117,-40.953,179.059,5.717,149.294
C03135=1178.258,-98.367,-40.944,179.058,5.717,149.294
C03136=1178.264,-98.617,-40.934,179.055,5.717,149.295
C03137=1178.269,-98.867,-40.925,179.053,5.717,149.295
C03138=1178.275,-99.116,-40.915,179.051,5.716,149.296
C03139=1178.279,-99.365,-40.905,179.049,5.716,149.297
C03140=1178.285,-99.616,-40.895,179.047,5.716,149.297
C03141=1178.290,-99.865,-40.886,179.045,5.716,149.298
C03142=1178.296,-100.116,-40.876,179.042,5.715,149.298
C03143=1178.300,-100.365,-40.867,179.040,5.715,149.299
C03144=1178.306,-100.615,-40.857,179.038,5.715,149.300
C03145=1178.311,-100.864,-40.847,179.036,5.714,149.300
C03146=1178.317,-101.114,-40.838,179.034,5.715,149.301
C03147=1178.321,-101.364,-40.828,179.032,5.714,149.301
C03148=1178.328,-101.636,-40.818,179.029,5.714,149.302
C03149=1178.334,-101.908,-40.807,179.027,5.714,149.303
C03150=1178.339,-102.179,-40.796,179.024,5.714,149.303
C03151=1178.344,-102.451,-40.786,179.022,5.713,149.304
C03152=1178.350,-102.701,-40.777,179.020,5.713,149.305
C03153=1178.355,-102.950,-40.767,179.018,5.712,149.305
C03154=1178.361,-103.201,-40.758,179.016,5.713,149.306
C03155=1178.366,-103.450,-40.748,179.013,5.712,149.306
C03156=1178.372,-103.700,-40.738,179.011,5.712,149.307
C03157=1178.377,-103.949,-40.729,179.009,5.712,149.308
C03158=1178.382,-104.199,-40.719,179.007,5.712,149.308
C03159=1178.387,-104.449,-40.710,179.005,5.711,149.309
C03160=1178.393,-104.698,-40.701,179.002,5.711,149.309
C03161=1178.398,-104.949,-40.691,179.001,5.711,149.310
C03162=1178.403,-105.199,-40.681,178.998,5.711,149.311
C03163=1178.409,-105.449,-40.672,178.996,5.711,149.311
C03164=1178.413,-105.698,-40.662,178.994,5.710,149.312
C03165=1178.419,-105.948,-40.653,178.992,5.710,149.312
C03166=1178.424,-106.197,-40.643,178.989,5.710,149.313
C03167=1178.429,-106.447,-40.634,178.988,5.710,149.314
C03168=1178.435,-106.697,-40.625,178.985,5.709,149.314
C03169=1178.440,-106.947,-40.615,178.983,5.709,149.315
C03170=1178.445,-107.196,-40.606,178.981,5.709,149.315
C03171=1178.451,-107.447,-40.597,178.979,5.708,149.316
C03172=1178.456,-107.696,-40.587,178.976,5.709,149.317
C03173=1178.462,-107.946,-40.578,178.974,5.708,149.317
C03174=1178.467,-108.195,-40.568,178.972,5.708,149.318
C03175=1178.472,-108.445,-40.559,178.970,5.708,149.318
C03176=1178.478,-108.695,-40.550,178.968,5.708,149.319
C03177=1178.483,-108.944,-40.540,178.966,5.707,149.320
C03178=1178.488,-109.194,-40.531,178.964,5.707,149.320
C03179=1178.494,-109.444,-40.522,178.961,5.707,149.321
C03180=1178.499,-109.694,-40.513,178.960,5.707,149.321
C03181=1178.504,-109.944,-40.503,178.957,5.706,149.322
C03182=1178.510,-110.194,-40.494,178.956,5.707,149.322
C03183=1178.515,-110.444,-40.485,178.953,5.706,149.323
C03184=1178.520,-110.693,-40.475,178.951,5.706,149.324
C03185=1178.526,-110.943,-40.466,178.949,5.706,149.324
C03186=1178.531,-111.193,-40.457,178.946,5.705,149.325
C03187=1178.536,-111.443,-40.448,178.944,5.705,149.326
C03188=1178.542,-111.692,-40.438,178.942,5.705,149.326
C03189=1178.547,-111.942,-40.429,178.940,5.705,149.327
C03190=1178.552,-112.192,-40.420,178.938,5.704,149.327
C03191=1178.557,-112.442,-40.411,178.936,5.704,149.328
C03192=1178.563,-112.691,-40.401,178.934,5.704,149.328
C03193=1178.568,-112.941,-40.392,178.932,5.704,149.329
C03194=1178.573,-113.191,-40.383,178.929,5.704,149.330
C03195=1178.579,-113.441,-40.373,178.928,5.704,149.330
C03196=1178.584,-113.690,-40.364,178.925,5.703,149.331
C03197=1178.589,-113.940,-40.355,178.923,5.703,149.331
C03198=1178.594,-114.190,-40.346,178.921,5.703,149.332
C03199=1178.600,-114.440,-40.337,178.919,5.703,149.333
C03200=1178.605,-114.690,-40.328,178.916,5.702,149.333
C03201=1178.610,-114.940,-40.319,178.915,5.702,149.334
C03202=1178.615,-115.189,-40.309,178.913,5.702,149.334
C03203=1178.622,-115.439,-40.300,178.911,5.702,149.335
C03204=1178.627,-115.688,-40.291,178.908,5.701,149.335
C03205=1178.632,-115.938,-40.282,178.906,5.702,149.336
C03206=1178.637,-116.188,-40.273,178.904,5.701,149.337
C03207=1178.643,-116.438,-40.264,178.902,5.701,149.337
C03208=1178.648,-116.688,-40.254,178.900,5.701,149.338
C03209=1178.653,-116.937,-40.245,178.898,5.701,149.338
C03210=1178.658,-117.187,-40.236,178.896,5.700,149.339
C03211=1178.664,-117.437,-40.228,178.894,5.700,149.339
C03212=1178.669,-117.687,-40.218,178.891,5.700,149.340
C03213=1178.675,-117.937,-40.209,178.890,5.700,149.341
C03214=1178.680,-118.186,-40.201,178.887,5.700,149.341
C03215=1178.686,-118.436,-40.192,178.885,5.700,149.342
C03216=1178.691,-118.686,-40.183,178.883,5.699,149.343
C03217=1178.696,-118.936,-40.174,178.881,5.699,149.343
C03218=1178.702,-119.186,-40.164,178.879,5.698,149.344
C03219=1178.707,-119.435,-40.155,178.877,5.699,149.344
C03220=1178.712,-119.685,-40.146,178.875,5.698,149.345
C03221=1178.717,-119.935,-40.137,178.873,5.699,149.346
C03222=1178.722,-120.185,-40.128,178.870,5.698,149.346
C03223=1178.728,-120.434,-40.120,178.869,5.698,149.346
C03224=1178.733,-120.684,-40.111,178.866,5.697,149.347
C03225=1178.738,-120.934,-40.102,178.865,5.697,149.348
C03226=1178.744,-121.184,-40.092,178.862,5.697,149.348
C03227=1178.749,-121.434,-40.083,178.860,5.697,149.349
C03228=1178.754,-121.684,-40.074,178.858,5.697,149.350
C03229=1178.760,-121.933,-40.066,178.856,5.697,149.350
C03230=1178.765,-122.183,-40.057,178.854,5.696,149.351
C03231=1178.771,-122.432,-40.048,178.852,5.696,149.351
C03232=1178.776,-122.682,-40.039,178.850,5.696,149.352
C03233=1178.781,-122.932,-40.030,178.847,5.696,149.352
C03234=1178.786,-123.182,-40.021,178.845,5.695,149.353
C03235=1178.792,-123.432,-40.012,178.844,5.695,149.353
C03236=1178.798,-123.681,-40.003,178.841,5.695,149.354
C03237=1178.803,-123.931,-39.995,178.839,5.695,149.355
C03238=1178.808,-124.182,-39.986,178.837,5.695,149.355
C03239=1178.814,-124.431,-39.977,178.835,5.695,149.356
C03240=1178.819,-124.681,-39.969,178.833,5.694,149.356
C03241=1178.824,-124.931,-39.960,178.831,5.694,149.357
C03242=1178.830,-125.180,-39.951,178.829,5.693,149.358
C03243=1178.835,-125.430,-39.942,178.827,5.694,149.358
C03244=1178.840,-125.680,-39.933,178.824,5.693,149.359
C03245=1178.845,-125.930,-39.924,178.823,5.693,149.359
C03246=1178.850,-126.180,-39.916,178.820,5.693,149.360
C03247=1178.856,-126.429,-39.907,178.818,5.693,149.360
C03248=1178.862,-126.679,-39.899,178.816,5.692,149.361
C03249=1178.867,-126.929,-39.890,178.814,5.692,149.362
C03250=1178.872,-127.179,-39.881,178.812,5.692,149.362
C03251=1178.877,-127.429,-39.872,178.810,5.692,149.363
C03252=1178.456,-127.439,-39.913,178.806,5.695,149.365
C03253=1178.451,-127.190,-39.921,178.809,5.696,149.364
C03254=1178.446,-126.940,-39.930,178.810,5.696,149.364
C03255=1178.440,-126.691,-39.939,178.812,5.696,149.363
C03256=1178.434,-126.440,-39.947,178.815,5.696,149.362
C03257=1178.429,-126.190,-39.956,178.817,5.697,149.362
C03258=1178.424,-125.940,-39.965,178.819,5.696,149.361
C03259=1178.419,-125.691,-39.974,178.820,5.696,149.361
C03260=1178.413,-125.441,-39.982,178.823,5.697,149.360
C03261=1178.408,-125.192,-39.991,178.825,5.697,149.359
C03262=1178.403,-124.942,-40.000,178.827,5.697,149.359
C03263=1178.398,-124.692,-40.009,178.829,5.697,149.358
C03264=1178.392,-124.442,-40.018,178.831,5.698,149.358
C03265=1178.387,-124.193,-40.026,178.833,5.698,149.357
C03266=1178.381,-123.943,-40.035,178.835,5.698,149.357
C03267=1178.376,-123.693,-40.043,178.837,5.698,149.356
C03268=1178.371,-123.443,-40.052,178.840,5.698,149.355
C03269=1178.366,-123.193,-40.061,178.841,5.698,149.355
C03270=1178.361,-122.943,-40.070,178.844,5.699,149.354
C03271=1178.354,-122.693,-40.079,178.846,5.699,149.354
C03272=1178.349,-122.444,-40.088,178.848,5.700,149.353
C03273=1178.344,-122.194,-40.097,178.850,5.699,149.352
C03274=1178.339,-121.944,-40.106,178.852,5.700,149.352
C03275=1178.333,-121.694,-40.115,178.854,5.700,149.351
C03276=1178.328,-121.444,-40.124,178.856,5.700,149.351
C03277=1178.322,-121.195,-40.132,178.858,5.700,149.350
C03278=1178.317,-120.945,-40.141,178.861,5.701,149.350
C03279=1178.312,-120.695,-40.150,178.862,5.701,149.349
C03280=1178.306,-120.445,-40.160,178.864,5.701,149.349
C03281=1178.301,-120.195,-40.169,178.867,5.701,149.348
C03282=1178.296,-119.946,-40.177,178.869,5.702,149.347
C03283=1178.291,-119.696,-40.186,178.871,5.701,149.347
C03284=1178.286,-119.446,-40.195,178.873,5.702,149.346
C03285=1178.280,-119.197,-40.204,178.875,5.702,149.346
C03286=1178.275,-118.947,-40.213,178.877,5.702,149.345
C03287=1178.269,-118.697,-40.223,178.879,5.702,149.344
C03288=1178.264,-118.447,-40.232,178.882,5.703,149.344
C03289=1178.259,-118.198,-40.241,178.883,5.703,149.343
C03290=1178.253,-117.948,-40.250,178.886,5.703,149.343
C03291=1178.248,-117.698,-40.258,178.887,5.703,149.342
C03292=1178.243,-117.448,-40.267,178.890,5.704,149.342
C03293=1178.237,-117.198,-40.277,178.892,5.703,149.341
C03294=1178.232,-116.948,-40.286,178.894,5.704,149.340
C03295=1178.226,-116.699,-40.294,178.896,5.704,149.340
C03296=1178.221,-116.449,-40.303,178.898,5.705,149.339
C03297=1178.216,-116.200,-40.313,178.900,5.704,149.338
C03298=1178.210,-115.950,-40.322,178.902,5.705,149.338
C03299=1178.205,-115.700,-40.331,178.904,5.705,149.337
C03300=1178.200,-115.450,-40.340,178.907,5.705,149.337
C03301=1178.195,-115.200,-40.349,178.908,5.705,149.336
C03302=1178.189,-114.950,-40.358,178.911,5.706,149.336
C03303=1178.184,-114.701,-40.368,178.913,5.706,149.335
C03304=1178.179,-114.451,-40.377,178.915,5.706,149.334
C03305=1178.174,-114.201,-40.386,178.917,5.706,149.334
C03306=1178.168,-113.951,-40.395,178.920,5.706,149.333
C03307=1178.163,-113.701,-40.404,178.921,5.706,149.333
C03308=1178.157,-113.452,-40.413,178.923,5.707,149.332
C03309=1178.152,-113.203,-40.422,178.926,5.708,149.331
C03310=1178.146,-112.952,-40.432,178.928,5.708,149.331
C03311=1178.141,-112.703,-40.441,178.930,5.708,149.330
C03312=1178.136,-112.453,-40.450,178.932,5.708,149.330
C03313=1178.131,-112.203,-40.459,178.935,5.708,149.329
C03314=1178.125,-111.953,-40.469,178.936,5.708,149.329
C03315=1178.120,-111.703,-40.478,178.939,5.709,149.328
C03316=1178.115,-111.454,-40.487,178.940,5.709,149.327
C03317=1178.109,-111.204,-40.497,178.943,5.709,149.327
C03318=1178.104,-110.954,-40.506,178.945,5.709,149.326
C03319=1178.099,-110.704,-40.515,178.947,5.710,149.326
C03320=1178.093,-110.454,-40.524,178.949,5.709,149.325
C03321=1178.088,-110.205,-40.534,178.951,5.710,149.325
C03322=1178.083,-109.955,-40.543,178.953,5.710,149.324
C03323=1178.077,-109.705,-40.552,178.955,5.710,149.323
C03324=1178.072,-109.456,-40.562,178.958,5.710,149.323
C03325=1178.067,-109.206,-40.571,178.960,5.711,149.322
C03326=1178.061,-108.956,-40.580,178.962,5.710,149.321
C03327=1178.056,-108.706,-40.590,178.964,5.711,149.321
C03328=1178.051,-108.457,-40.599,178.967,5.712,149.320
C03329=1178.045,-108.206,-40.608,178.968,5.712,149.320
C03330=1178.040,-107.957,-40.618,178.971,5.712,149.319
C03331=1178.035,-107.707,-40.627,178.973,5.712,149.319
C03332=1178.029,-107.457,-40.636,178.975,5.712,149.318
C03333=1178.024,-107.208,-40.646,178.977,5.712,149.317
C03334=1178.018,-106.958,-40.655,178.979,5.713,149.317
C03335=1178.013,-106.708,-40.664,178.981,5.713,149.316
C03336=1178.008,-106.459,-40.674,178.983,5.713,149.316
C03337=1178.003,-106.208,-40.684,178.985,5.713,149.315
C03338=1177.998,-105.959,-40.693,178.988,5.714,149.314
C03339=1177.993,-105.709,-40.702,178.990,5.713,149.314
C03340=1177.987,-105.459,-40.712,178.992,5.714,149.313
C03341=1177.982,-105.209,-40.721,178.995,5.715,149.313
C03342=1177.976,-104.959,-40.731,178.996,5.715,149.312
C03343=1177.972,-104.710,-40.740,178.999,5.715,149.311
C03344=1177.966,-104.460,-40.750,179.000,5.715,149.311
C03345=1177.960,-104.210,-40.759,179.003,5.715,149.310
C03346=1177.956,-103.961,-40.768,179.005,5.715,149.310
C03347=1177.950,-103.711,-40.778,179.007,5.716,149.309
C03348=1177.945,-103.461,-40.787,179.009,5.716,149.308
C03349=1177.939,-103.211,-40.797,179.012,5.716,149.308
C03350=1177.934,-102.962,-40.807,179.014,5.717,149.307
C03351=1177.929,-102.711,-40.816,179.016,5.716,149.307
C03352=1177.924,-102.462,-40.826,179.018,5.717,149.306
C03353=1177.918,-102.191,-40.836,179.020,5.717,149.305
C03354=1177.912,-101.918,-40.847,179.023,5.717,149.305
C03355=1177.906,-101.646,-40.857,179.025,5.718,149.304
C03356=1177.901,-101.375,-40.868,179.027,5.718,149.303
C03357=1177.895,-101.125,-40.877,179.030,5.718,149.303
C03358=1177.890,-100.876,-40.887,179.032,5.719,149.302
C03359=1177.884,-100.626,-40.896,179.034,5.718,149.302
C03360=1177.879,-100.376,-40.906,179.036,5.719,149.301
C03361=1177.873,-100.126,-40.916,179.038,5.719,149.300
C03362=1177.869,-99.876,-40.926,179.041,5.719,149.300
C03363=1177.863,-99.626,-40.935,179.043,5.719,149.299
C03364=1177.858,-99.377,-40.945,179.045,5.720,149.299
C03365=1177.853,-99.127,-40.955,179.047,5.719,149.298
C03366=1177.848,-98.878,-40.964,179.049,5.720,149.297
C03367=1177.842,-98.628,-40.974,179.052,5.721,149.297
C03368=1177.837,-98.378,-40.983,179.053,5.721,149.296
C03369=1177.831,-98.129,-40.993,179.056,5.721,149.296
C03370=1177.827,-97.879,-41.003,179.058,5.721,149.295
C03371=1177.821,-97.628,-41.013,179.060,5.721,149.294
C03372=1177.816,-97.379,-41.023,179.062,5.721,149.294
C03373=1177.810,-97.129,-41.032,179.065,5.722,149.293
C03374=1177.805,-96.880,-41.042,179.067,5.723,149.293
C03375=1177.800,-96.630,-41.051,179.069,5.722,149.292
C03376=1177.795,-96.379,-41.061,179.071,5.723,149.291
C03377=1177.789,-96.130,-41.072,179.073,5.723,149.291
C03378=1177.784,-95.881,-41.081,179.075,5.723,149.290
C03379=1177.778,-95.631,-41.091,179.077,5.723,149.290
C03380=1177.773,-95.381,-41.100,179.080,5.724,149.289
C03381=1177.768,-95.131,-41.111,179.082,5.724,149.288
C03382=1177.763,-94.881,-41.120,179.084,5.724,149.288
C03383=1177.758,-94.632,-41.130,179.087,5.724,149.287
C03384=1177.752,-94.382,-41.140,179.088,5.724,149.287
C03385=1177.746,-94.132,-41.150,179.091,5.725,149.286
C03386=1177.742,-93.882,-41.160,179.093,5.725,149.285
C03387=1177.736,-93.632,-41.170,179.095,5.725,149.285
C03388=1177.731,-93.383,-41.179,179.098,5.726,149.284
C03389=1177.726,-93.133,-41.189,179.099,5.726,149.284
C03390=1177.720,-92.884,-41.199,179.102,5.726,149.283
C03391=1177.716,-92.634,-41.209,179.104,5.727,149.282
C03392=1177.710,-92.384,-41.219,179.106,5.726,149.282
C03393=1177.704,-92.134,-41.229,179.108,5.727,149.281
C03394=1177.699,-91.885,-41.238,179.111,5.727,149.280
C03395=1177.694,-91.634,-41.249,179.113,5.728,149.280
C03396=1177.689,-91.385,-41.259,179.115,5.727,149.279
C03397=1177.684,-91.136,-41.269,179.117,5.728,149.279
C03398=1177.678,-90.885,-41.278,179.120,5.728,149.278
C03399=1177.672,-90.636,-41.289,179.121,5.728,149.278
C03400=1177.667,-90.386,-41.299,179.124,5.729,149.277
C03401=1177.662,-90.136,-41.309,179.126,5.728,149.276
C03402=1177.657,-89.887,-41.319,179.128,5.729,149.276
C03403=1177.652,-89.636,-41.329,179.131,5.729,149.275
C03404=1177.647,-89.387,-41.338,179.133,5.729,149.275
C03405=1177.641,-89.137,-41.349,179.135,5.730,149.274
C03406=1177.636,-88.888,-41.359,179.137,5.730,149.273
C03407=1177.631,-88.637,-41.369,179.139,5.730,149.273
C03408=1177.626,-88.388,-41.379,179.142,5.731,149.272
C03409=1177.620,-88.139,-41.389,179.144,5.731,149.271
C03410=1177.614,-87.889,-41.399,179.146,5.731,149.271
C03411=1177.609,-87.638,-41.409,179.148,5.731,149.270
C03412=1177.604,-87.389,-41.419,179.151,5.731,149.270
C03413=1177.599,-87.140,-41.429,179.153,5.732,149.269
C03414=1177.594,-86.889,-41.440,179.155,5.732,149.268
C03415=1177.588,-86.640,-41.450,179.157,5.733,149.268
C03416=1177.583,-86.391,-41.459,179.160,5.733,149.267
C03417=1177.578,-86.140,-41.470,179.161,5.733,149.267
C03418=1177.573,-85.891,-41.480,179.164,5.733,149.266
C03419=1177.567,-85.641,-41.490,179.166,5.733,149.265
C03420=1177.562,-85.391,-41.501,179.168,5.734,149.265
C03421=1177.557,-85.142,-41.511,179.171,5.734,149.264
C03422=1177.552,-84.892,-41.521,179.173,5.734,149.264
C03423=1177.547,-84.642,-41.531,179.175,5.735,149.263
C03424=1177.541,-84.392,-41.542,179.177,5.735,149.262
C03425=1177.535,-84.143,-41.552,179.180,5.735,149.262
C03426=1177.531,-83.893,-41.562,179.182,5.736,149.261
C03427=1177.526,-83.643,-41.572,179.184,5.735,149.260
C03428=1177.520,-83.394,-41.582,179.186,5.736,149.260
C03429=1177.515,-83.144,-41.593,179.189,5.737,149.259
C03430=1177.509,-82.894,-41.603,179.191,5.736,149.259
C03431=1177.504,-82.644,-41.613,179.193,5.737,149.258
C03432=1177.499,-82.394,-41.624,179.195,5.737,149.257
C03433=1177.494,-82.145,-41.633,179.197,5.737,149.257
C03434=1177.488,-81.895,-41.644,179.200,5.738,149.256
C03435=1177.483,-81.645,-41.654,179.201,5.738,149.256
C03436=1177.478,-81.396,-41.664,179.204,5.738,149.255
C03437=1177.473,-81.145,-41.675,179.207,5.739,149.254
C03438=1177.467,-80.896,-41.685,179.208,5.739,149.254
C03439=1177.462,-80.646,-41.695,179.211,5.739,149.253
C03440=1177.457,-80.396,-41.706,179.213,5.740,149.253
C03441=1177.451,-80.147,-41.716,179.215,5.739,149.252
C03442=1177.447,-79.897,-41.726,179.218,5.740,149.251
C03443=1177.441,-79.648,-41.737,179.220,5.740,149.251
C03444=1177.436,-79.398,-41.747,179.222,5.740,149.250
C03445=1177.431,-79.148,-41.758,179.225,5.741,149.250
C03446=1177.425,-78.898,-41.768,179.227,5.741,149.249
C03447=1177.420,-78.648,-41.779,179.229,5.741,149.248
C03448=1177.415,-78.399,-41.789,179.231,5.742,149.248
C03449=1177.409,-78.149,-41.799,179.233,5.742,149.247
C03450=1177.404,-77.899,-41.810,179.236,5.742,149.246
C03451=1177.399,-77.650,-41.821,179.238,5.743,149.246
C03452=1177.394,-77.400,-41.831,179.240,5.743,149.245
C03453=1177.388,-77.150,-41.841,179.243,5.743,149.245
C03454=1177.383,-76.900,-41.852,179.245,5.744,149.244
C03455=1177.377,-76.650,-41.862,179.247,5.743,149.243
C03456=1177.372,-76.401,-41.873,179.250,5.744,149.243
C03457=1177.367,-76.130,-41.884,179.252,5.745,149.242
C03458=1177.361,-75.858,-41.896,179.254,5.744,149.241
C03459=1177.355,-75.588,-41.907,179.257,5.745,149.241
C03460=1177.350,-75.317,-41.918,179.259,5.745,149.240
C03461=1177.344,-75.067,-41.929,179.261,5.746,149.240
C03462=1177.339,-74.818,-41.940,179.263,5.745,149.239
C03463=1177.334,-74.568,-41.950,179.266,5.746,149.238
C03464=1177.329,-74.318,-41.961,179.268,5.747,149.238
C03465=1177.323,-74.068,-41.971,179.270,5.746,149.237
C03466=1177.319,-73.819,-41.982,179.273,5.747,149.236
C03467=1177.313,-73.569,-41.992,179.275,5.747,149.236
C03468=1177.308,-73.319,-42.003,179.277,5.747,149.235
C03469=1177.302,-73.069,-42.014,179.280,5.748,149.235
C03470=1177.297,-72.819,-42.025,179.282,5.748,149.234
C03471=1177.291,-72.570,-42.035,179.284,5.748,149.233
C03472=1177.286,-72.320,-42.046,179.286,5.749,149.233
C03473=1177.281,-72.071,-42.057,179.289,5.749,149.232
C03474=1177.276,-71.821,-42.067,179.291,5.749,149.231
C03475=1177.270,-71.571,-42.078,179.293,5.749,149.231
C03476=1177.266,-71.321,-42.089,179.296,5.750,149.230
C03477=1177.260,-71.072,-42.099,179.298,5.750,149.230
C03478=1177.255,-70.822,-42.110,179.300,5.751,149.229
C03479=1177.250,-70.573,-42.121,179.303,5.751,149.228
C03480=1177.244,-70.322,-42.132,179.305,5.751,149.228
C03481=1177.238,-70.073,-42.142,179.307,5.751,149.227
C03482=1177.234,-69.823,-42.153,179.309,5.752,149.226
C03483=1177.228,-69.573,-42.163,179.311,5.752,149.226
C03484=1177.224,-69.324,-42.175,179.314,5.752,149.225
C03485=1177.218,-69.074,-42.185,179.316,5.753,149.225
C03486=1177.213,-68.825,-42.196,179.318,5.753,149.224
C03487=1177.208,-68.574,-42.207,179.321,5.753,149.223
C03488=1177.202,-68.324,-42.218,179.323,5.754,149.223
C03489=1177.197,-68.075,-42.229,179.325,5.754,149.222
C03490=1177.192,-67.825,-42.239,179.328,5.754,149.222
C03491=1177.187,-67.576,-42.250,179.330,5.755,149.221
C03492=1177.181,-67.326,-42.261,179.332,5.755,149.220
C03493=1177.177,-67.077,-42.272,179.335,5.755,149.220
C03494=1177.170,-66.827,-42.283,179.337,5.756,149.219
C03495=1177.166,-66.577,-42.294,179.339,5.756,149.218
C03496=1177.161,-66.327,-42.305,179.341,5.756,149.218
C03497=1177.155,-66.078,-42.315,179.344,5.756,149.217
C03498=1177.150,-65.828,-42.326,179.346,5.757,149.217
C03499=1177.144,-65.578,-42.338,179.348,5.757,149.216
C03500=1177.139,-65.328,-42.348,179.351,5.757,149.215
C03501=1177.135,-65.079,-42.359,179.353,5.758,149.215
C03502=1177.129,-64.829,-42.370,179.355,5.758,149.214
C03503=1177.124,-64.579,-42.381,179.358,5.758,149.213
C03504=1177.118,-64.330,-42.392,179.360,5.759,149.213
C03505=1177.113,-64.080,-42.403,179.362,5.759,149.212
C03506=1177.108,-63.830,-42.414,179.364,5.759,149.212
C03507=1177.103,-63.581,-42.425,179.367,5.760,149.211
C03508=1177.097,-63.330,-42.436,179.369,5.760,149.210
C03509=1177.093,-63.081,-42.447,179.371,5.760,149.210
C03510=1177.087,-62.832,-42.458,179.374,5.760,149.209
C03511=1177.082,-62.581,-42.468,179.376,5.761,149.209
C03512=1177.076,-62.332,-42.480,179.378,5.761,149.208
C03513=1177.071,-62.082,-42.491,179.380,5.761,149.207
C03514=1177.067,-61.832,-42.502,179.383,5.762,149.207
C03515=1177.061,-61.583,-42.513,179.385,5.763,149.206
C03516=1177.055,-61.333,-42.524,179.387,5.762,149.205
C03517=1177.051,-61.083,-42.535,179.390,5.763,149.205
C03518=1177.046,-60.834,-42.546,179.392,5.763,149.204
C03519=1177.040,-60.584,-42.557,179.394,5.763,149.204
C03520=1177.035,-60.334,-42.569,179.397,5.764,149.203
C03521=1177.030,-60.085,-42.580,179.399,5.764,149.202
C03522=1177.024,-59.835,-42.591,179.401,5.765,149.202
C03523=1177.019,-59.585,-42.602,179.403,5.765,149.201
C03524=1177.014,-59.336,-42.613,179.406,5.765,149.200
C03525=1177.008,-59.085,-42.624,179.408,5.766,149.200
C03526=1177.004,-58.836,-42.635,179.411,5.766,149.199
C03527=1176.998,-58.587,-42.646,179.413,5.766,149.199
C03528=1176.993,-58.337,-42.658,179.415,5.767,149.198
C03529=1176.988,-58.087,-42.669,179.418,5.767,149.197
C03530=1176.983,-57.837,-42.680,179.420,5.767,149.197
C03531=1176.977,-57.588,-42.692,179.422,5.768,149.196
C03532=1176.972,-57.338,-42.702,179.425,5.768,149.196
C03533=1176.968,-57.088,-42.713,179.427,5.769,149.195
C03534=1176.961,-56.839,-42.725,179.429,5.768,149.194
C03535=1176.957,-56.589,-42.736,179.432,5.769,149.194
C03536=1176.951,-56.339,-42.748,179.434,5.770,149.193
C03537=1176.946,-56.089,-42.759,179.437,5.770,149.192
C03538=1176.941,-55.840,-42.770,179.438,5.770,149.192
C03539=1176.936,-55.590,-42.782,179.441,5.770,149.191
C03540=1176.931,-55.340,-42.793,179.444,5.771,149.191
C03541=1176.926,-55.091,-42.805,179.445,5.771,149.190
C03542=1176.920,-54.841,-42.815,179.448,5.771,149.189
C03543=1176.915,-54.591,-42.826,179.450,5.772,149.189
C03544=1176.910,-54.341,-42.838,179.453,5.773,149.188
C03545=1176.905,-54.092,-42.849,179.455,5.772,149.188
C03546=1176.899,-53.843,-42.861,179.457,5.773,149.187
C03547=1176.894,-53.593,-42.872,179.460,5.773,149.186
C03548=1176.889,-53.343,-42.884,179.462,5.774,149.186
C03549=1176.884,-53.093,-42.895,179.464,5.774,149.185
C03550=1176.878,-52.844,-42.906,179.467,5.774,149.184
C03551=1176.873,-52.594,-42.917,179.469,5.775,149.184
C03552=1176.869,-52.344,-42.929,179.471,5.775,149.183
C03553=1176.863,-52.094,-42.941,179.473,5.775,149.183
C03554=1176.858,-51.845,-42.952,179.476,5.776,149.182
C03555=1176.852,-51.595,-42.963,179.478,5.776,149.181
C03556=1176.848,-51.346,-42.975,179.481,5.777,149.181
C03557=1176.842,-51.096,-42.987,179.483,5.776,149.180
C03558=1176.838,-50.846,-42.998,179.485,5.777,149.179
C03559=1176.832,-50.596,-43.010,179.488,5.778,149.179
C03560=1176.826,-50.346,-43.021,179.490,5.778,149.178
C03561=1176.821,-50.076,-43.033,179.493,5.779,149.178
C03562=1176.816,-49.806,-43.046,179.495,5.779,149.177
C03563=1176.810,-49.536,-43.058,179.497,5.779,149.176
C03564=1176.804,-49.265,-43.071,179.500,5.779,149.175
C03565=1176.799,-49.016,-43.083,179.503,5.780,149.175
C03566=1176.794,-48.766,-43.094,179.505,5.781,149.174
C03567=1176.788,-48.517,-43.105,179.508,5.781,149.174
C03568=1176.783,-48.267,-43.117,179.509,5.781,149.173
C03569=1176.778,-48.017,-43.129,179.512,5.781,149.172
C03570=1176.773,-47.767,-43.141,179.515,5.782,149.172
C03571=1176.768,-47.518,-43.152,179.517,5.783,149.171
C03572=1176.763,-47.268,-43.164,179.519,5.783,149.171
C03573=1176.757,-47.018,-43.175,179.522,5.783,149.170
C03574=1176.752,-46.769,-43.187,179.524,5.784,149.169
C03575=1176.746,-46.519,-43.198,179.526,5.784,149.169
C03576=1176.742,-46.269,-43.210,179.529,5.784,149.168
C03577=1176.736,-46.019,-43.222,179.531,5.784,149.168
C03578=1176.731,-45.769,-43.233,179.533,5.785,149.167
C03579=1176.726,-45.520,-43.245,179.536,5.785,149.166
C03580=1176.720,-45.270,-43.256,179.538,5.786,149.166
C03581=1176.716,-45.021,-43.268,179.541,5.786,149.165
C03582=1176.710,-44.772,-43.280,179.543,5.786,149.164
C03583=1176.705,-44.522,-43.292,179.545,5.787,149.164
C03584=1176.700,-44.272,-43.303,179.548,5.787,149.163
C03585=1176.695,-44.022,-43.315,179.550,5.788,149.163
C03586=1176.689,-43.772,-43.327,179.552,5.788,149.162
C03587=1176.685,-43.522,-43.338,179.555,5.788,149.161
C03588=1176.680,-43.273,-43.351,179.557,5.789,149.161
C03589=1176.674,-43.023,-43.363,179.559,5.789,149.160
C03590=1176.669,-42.774,-43.374,179.562,5.790,149.159
C03591=1176.663,-42.524,-43.386,179.564,5.790,149.159
C03592=1176.658,-42.274,-43.398,179.566,5.790,149.158
C03593=1176.653,-42.025,-43.410,179.569,5.791,149.157
C03594=1176.648,-41.775,-43.421,179.571,5.792,149.157
C03595=1176.643,-41.526,-43.433,179.574,5.792,149.156
C03596=1176.637,-41.276,-43.445,179.576,5.792,149.156
C03597=1176.633,-41.026,-43.457,179.578,5.792,149.155
C03598=1176.627,-40.777,-43.469,179.581,5.793,149.154
C03599=1176.622,-40.527,-43.481,179.584,5.793,149.154
C03600=1176.617,-40.277,-43.493,179.586,5.794,149.153
C03601=1176.612,-40.027,-43.504,179.588,5.794,149.152
C03602=1176.607,-39.778,-43.517,179.590,5.794,149.152
C03603=1176.601,-39.528,-43.529,179.593,5.795,149.151
C03604=1176.596,-39.278,-43.541,179.595,5.795,149.151
C03605=1176.592,-39.029,-43.553,179.598,5.796,149.150
C03606=1176.586,-38.779,-43.564,179.600,5.797,149.149
C03607=1176.581,-38.529,-43.576,179.602,5.796,149.149
C03608=1176.576,-38.280,-43.589,179.605,5.797,149.148
C03609=1176.570,-38.030,-43.601,179.607,5.798,149.148
C03610=1176.565,-37.780,-43.612,179.610,5.798,149.147
C03611=1176.560,-37.531,-43.625,179.612,5.799,149.146
C03612=1176.555,-37.281,-43.637,179.614,5.798,149.146
C03613=1176.549,-37.031,-43.648,179.617,5.799,149.145
C03614=1176.544,-36.782,-43.661,179.619,5.800,149.145
C03615=1176.540,-36.532,-43.672,179.621,5.800,149.144
C03616=1176.534,-36.282,-43.684,179.624,5.801,149.143
C03617=1176.529,-36.033,-43.697,179.626,5.801,149.143
C03618=1176.524,-35.783,-43.709,179.628,5.801,149.142
C03619=1176.518,-35.533,-43.721,179.631,5.802,149.141
C03620=1176.513,-35.284,-43.733,179.633,5.802,149.141
C03621=1176.508,-35.034,-43.745,179.636,5.803,149.140
C03622=1176.503,-34.785,-43.757,179.639,5.803,149.139
C03623=1176.498,-34.535,-43.769,179.641,5.804,149.139
C03624=1176.493,-34.285,-43.782,179.643,5.804,149.138
C03625=1176.487,-34.035,-43.794,179.645,5.804,149.138
C03626=1176.482,-33.786,-43.806,179.648,5.805,149.137
C03627=1176.477,-33.536,-43.818,179.650,5.805,149.136
C03628=1176.471,-33.286,-43.830,179.653,5.806,149.136
C03629=1176.466,-33.037,-43.842,179.655,5.807,149.135
C03630=1176.462,-32.787,-43.854,179.657,5.806,149.134
C03631=1176.456,-32.538,-43.866,179.660,5.807,149.134
C03632=1176.451,-32.288,-43.878,179.662,5.808,149.133
C03633=1176.446,-32.039,-43.891,179.665,5.808,149.133
C03634=1176.440,-31.789,-43.903,179.667,5.808,149.132
C03635=1176.435,-31.540,-43.915,179.670,5.809,149.131
C03636=1176.430,-31.290,-43.928,179.672,5.809,149.131
C03637=1176.425,-31.040,-43.940,179.674,5.809,149.130
C03638=1176.420,-30.790,-43.953,179.676,5.810,149.130
C03639=1176.415,-30.540,-43.965,179.679,5.811,149.129
C03640=1176.410,-30.291,-43.977,179.682,5.811,149.128
C03641=1176.404,-30.041,-43.989,179.684,5.812,149.128
C03642=1176.399,-29.792,-44.002,179.687,5.812,149.127
C03643=1176.394,-29.542,-44.014,179.689,5.812,149.126
C03644=1176.389,-29.292,-44.026,179.691,5.813,149.126
C03645=1176.383,-29.043,-44.039,179.694,5.813,149.125
C03646=1176.379,-28.793,-44.051,179.696,5.814,149.124
C03647=1176.373,-28.543,-44.064,179.698,5.814,149.124
C03648=1176.368,-28.294,-44.076,179.701,5.815,149.123
